LIN {X 0,Y 614.5,Z 958.979,A -85,B 0,C 180,E1 26505.989,E2 26505.989} C_VEL
LIN {X 0,Y 616.34,Z 935.943,A -85,B 0,C 180,E1 26505.389,E2 26505.389} C_VEL
LIN {X 0,Y 618.103,Z 906.869,A -85,B 0,C 180,E1 26504.819,E2 26504.819} C_VEL
LIN {X 0,Y 619.74,Z 852.233,A -85,B 0,C 180,E1 26504.043,E2 26504.043} C_VEL
LIN {X 0,Y 625.607,Z 633.811,A -85,B 0,C 180,E1 26500.991,E2 26500.991} C_VEL
LIN {X 0,Y 629.765,Z 486.938,A -85,B 0,C 180,E1 26498.889,E2 26498.889} C_VEL
LIN {X 0,Y 615.789,Z 466.074,A -85,B 0,C 180,E1 26496.868,E2 26496.868} C_VEL
LIN {X 0,Y 606.821,Z 453.224,A -85,B 0,C 180,E1 26495.48,E2 26495.48} C_VEL
LIN {X 0,Y 598.746,Z 442.127,A -85,B 0,C 180,E1 26494.162,E2 26494.162} C_VEL
LIN {X 0,Y 588.904,Z 428.967,A -85,B 0,C 180,E1 26492.448,E2 26492.448} C_VEL
LIN {X 0,Y 585.376,Z 424.275,A -85,B 0,C 180,E1 26491.8,E2 26491.8} C_VEL
LIN {X 0,Y 583.558,Z 421.917,A -85,B 0,C 180,E1 26491.392,E2 26491.392} C_VEL
LIN {X 0,Y 582.067,Z 418.761,A -85,B 0,C 180,E1 26490.791,E2 26490.791} C_VEL
LIN {X 0,Y 580.207,Z 415.439,A -85,B 0,C 180,E1 26490.099,E2 26490.099} C_VEL
LIN {X 0,Y 579.523,Z 413.86,A -85,B 0,C 180,E1 26489.796,E2 26489.796} C_VEL
LIN {X 0,Y 577.505,Z 410.525,A -85,B 0,C 180,E1 26489.047,E2 26489.047} C_VEL
LIN {X 0,Y 577.246,Z 409.292,A -85,B 0,C 180,E1 26488.795,E2 26488.795} C_VEL
LIN {X 0,Y 577.307,Z 409.275,A -85,B 0,C 180,E1 26485.658,E2 26485.658} C_VEL
LIN {X 0,Y 577.239,Z 409.328,A -85,B 0,C 180,E1 26482.613,E2 26482.613} C_VEL
LIN {X 0,Y 577.304,Z 409.276,A -85,B 0,C 180,E1 26479.529,E2 26479.529} C_VEL
LIN {X 0,Y 577.227,Z 409.31,A -85,B 0,C 180,E1 26476.504,E2 26476.504} C_VEL
LIN {X 0,Y 577.301,Z 409.291,A -85,B 0,C 180,E1 26473.42,E2 26473.42} C_VEL
LIN {X 0,Y 577.214,Z 409.295,A -85,B 0,C 180,E1 26470.278,E2 26470.278} C_VEL
LIN {X 0,Y 577.279,Z 409.308,A -85,B 0,C 180,E1 26467.097,E2 26467.097} C_VEL
LIN {X 0,Y 577.215,Z 409.289,A -85,B 0,C 180,E1 26464.073,E2 26464.073} C_VEL
LIN {X 0,Y 577.286,Z 409.311,A -85,B 0,C 180,E1 26460.893,E2 26460.893} C_VEL
LIN {X 0,Y 577.226,Z 409.286,A -85,B 0,C 180,E1 26457.915,E2 26457.915} C_VEL
LIN {X 0,Y 577.293,Z 409.312,A -85,B 0,C 180,E1 26454.733,E2 26454.733} C_VEL
LIN {X 0,Y 577.237,Z 409.283,A -85,B 0,C 180,E1 26451.734,E2 26451.734} C_VEL
LIN {X 0,Y 577.296,Z 409.318,A -85,B 0,C 180,E1 26448.511,E2 26448.511} C_VEL
LIN {X 0,Y 577.25,Z 409.278,A -85,B 0,C 180,E1 26445.454,E2 26445.454} C_VEL
LIN {X 0,Y 577.285,Z 409.321,A -85,B 0,C 180,E1 26442.147,E2 26442.147} C_VEL
LIN {X 0,Y 577.272,Z 409.275,A -85,B 0,C 180,E1 26439.095,E2 26439.095} C_VEL
LIN {X 0,Y 577.272,Z 409.3,A -85,B 0,C 180,E1 26435.763,E2 26435.763} C_VEL
LIN {X 0,Y 577.315,Z 409.306,A -85,B 0,C 180,E1 26432.567,E2 26432.567} C_VEL
LIN {X 0,Y 577.279,Z 409.351,A -85,B 0,C 180,E1 26429.358,E2 26429.358} C_VEL
LIN {X 0,Y 578.244,Z 412.23,A -85,B 0,C 180,E1 26429.127,E2 26429.127} C_VEL
LIN {X 0,Y 580.66,Z 414.858,A -85,B 0,C 180,E1 26428.665,E2 26428.665} C_VEL
LIN {X 0,Y 582.281,Z 416.079,A -85,B 0,C 180,E1 26428.373,E2 26428.373} C_VEL
LIN {X 0,Y 584.579,Z 419.788,A -85,B 0,C 180,E1 26427.92,E2 26427.92} C_VEL
LIN {X 0,Y 587.298,Z 422.366,A -85,B 0,C 180,E1 26427.438,E2 26427.438} C_VEL
LIN {X 0,Y 590.315,Z 426.389,A -85,B 0,C 180,E1 26426.889,E2 26426.889} C_VEL
LIN {X 0,Y 592.156,Z 428.364,A -85,B 0,C 180,E1 26426.572,E2 26426.572} C_VEL
LIN {X 0,Y 595.83,Z 432.899,A -85,B 0,C 180,E1 26425.938,E2 26425.938} C_VEL
LIN {X 0,Y 602.194,Z 441.085,A -85,B 0,C 180,E1 26424.877,E2 26424.877} C_VEL
LIN {X 0,Y 609.795,Z 450.687,A -85,B 0,C 180,E1 26423.676,E2 26423.676} C_VEL
LIN {X 0,Y 621.483,Z 466.359,A -85,B 0,C 180,E1 26421.931,E2 26421.931} C_VEL
LIN {X 0,Y 629.591,Z 477.801,A -85,B 0,C 180,E1 26420.786,E2 26420.786} C_VEL
LIN {X 0,Y 623.132,Z 702.195,A -85,B 0,C 180,E1 26417.599,E2 26417.599} C_VEL
LIN {X 0,Y 622.882,Z 711.323,A -85,B 0,C 180,E1 26417.471,E2 26417.471} C_VEL
LIN {X 0,Y 621.995,Z 719.027,A -85,B 0,C 180,E1 26417.431,E2 26417.431} C_VEL
LIN {X 0,Y 617.19,Z 739.673,A -85,B 0,C 180,E1 26417.572,E2 26417.572} C_VEL
LIN {X 0,Y 616.501,Z 746.282,A -85,B 0,C 180,E1 26417.53,E2 26417.53} C_VEL
LIN {X 0,Y 612.714,Z 875.215,A -85,B 0,C 180,E1 26415.71,E2 26415.71} C_VEL
LIN {X 0,Y 611.293,Z 900.177,A -85,B 0,C 180,E1 26415.25,E2 26415.25} C_VEL
LIN {X 0,Y 609.06,Z 927.879,A -85,B 0,C 180,E1 26414.552,E2 26414.552} C_VEL
LIN {X 0,Y 606.986,Z 949.44,A -85,B 0,C 180,E1 26413.867,E2 26413.867} C_VEL
LIN {X 0,Y 604.786,Z 969.358,A -85,B 0,C 180,E1 26413.119,E2 26413.119} C_VEL
LIN {X 0,Y 602.352,Z 989.561,A -85,B 0,C 180,E1 26412.235,E2 26412.235} C_VEL
LIN {X 0,Y 599.698,Z 1009.452,A -85,B 0,C 180,E1 26411.239,E2 26411.239} C_VEL
LIN {X 0,Y 596.122,Z 1034.235,A -85,B 0,C 180,E1 26409.806,E2 26409.806} C_VEL
LIN {X 0,Y 592.792,Z 1055.848,A -85,B 0,C 180,E1 26408.361,E2 26408.361} C_VEL
LIN {X 0,Y 589.917,Z 1074.13,A -85,B 0,C 180,E1 26406.985,E2 26406.985} C_VEL
LIN {X 0,Y 587.066,Z 1091.868,A -85,B 0,C 180,E1 26405.498,E2 26405.498} C_VEL
LIN {X 0,Y 583.798,Z 1112.341,A -85,B 0,C 180,E1 26403.58,E2 26403.58} C_VEL
LIN {X 0,Y 580.752,Z 1131.299,A -85,B 0,C 180,E1 26401.542,E2 26401.542} C_VEL
LIN {X 0,Y 578.394,Z 1146.388,A -85,B 0,C 180,E1 26399.738,E2 26399.738} C_VEL
LIN {X 0,Y 576.222,Z 1160.882,A -85,B 0,C 180,E1 26397.819,E2 26397.819} C_VEL
LIN {X 0,Y 573.962,Z 1177.393,A -85,B 0,C 180,E1 26395.369,E2 26395.369} C_VEL
LIN {X 0,Y 572.132,Z 1191.681,A -85,B 0,C 180,E1 26392.924,E2 26392.924} C_VEL
LIN {X 0,Y 570.833,Z 1203.133,A -85,B 0,C 180,E1 26390.711,E2 26390.711} C_VEL
LIN {X 0,Y 569.76,Z 1214.119,A -85,B 0,C 180,E1 26388.3,E2 26388.3} C_VEL
LIN {X 0,Y 568.912,Z 1224.958,A -85,B 0,C 180,E1 26385.489,E2 26385.489} C_VEL
LIN {X 0,Y 568.45,Z 1232.629,A -85,B 0,C 180,E1 26383.11,E2 26383.11} C_VEL
LIN {X 0,Y 568.167,Z 1238.465,A -85,B 0,C 180,E1 26380.951,E2 26380.951} C_VEL
LIN {X 0,Y 568.021,Z 1243.665,A -85,B 0,C 180,E1 26378.6,E2 26378.6} C_VEL
LIN {X 0,Y 567.937,Z 1248.127,A -85,B 0,C 180,E1 26375.856,E2 26375.856} C_VEL
LIN {X 0,Y 567.911,Z 1250.647,A -85,B 0,C 180,E1 26373.326,E2 26373.326} C_VEL
LIN {X 0,Y 567.894,Z 1251.727,A -85,B 0,C 180,E1 26371.206,E2 26371.206} C_VEL
LIN {X 0,Y 567.865,Z 1251.836,A -85,B 0,C 180,E1 26369.188,E2 26369.188} C_VEL
LIN {X 0,Y 567.909,Z 1250.974,A -85,B 0,C 180,E1 26367.069,E2 26367.069} C_VEL
LIN {X 0,Y 567.923,Z 1249.038,A -85,B 0,C 180,E1 26364.844,E2 26364.844} C_VEL
LIN {X 0,Y 567.957,Z 1245.803,A -85,B 0,C 180,E1 26362.51,E2 26362.51} C_VEL
LIN {X 0,Y 568.095,Z 1240.685,A -85,B 0,C 180,E1 26359.859,E2 26359.859} C_VEL
LIN {X 0,Y 568.383,Z 1233.775,A -85,B 0,C 180,E1 26357.19,E2 26357.19} C_VEL
LIN {X 0,Y 568.807,Z 1226.648,A -85,B 0,C 180,E1 26354.916,E2 26354.916} C_VEL
LIN {X 0,Y 569.369,Z 1218.647,A -85,B 0,C 180,E1 26352.732,E2 26352.732} C_VEL
LIN {X 0,Y 570.319,Z 1208.371,A -85,B 0,C 180,E1 26350.302,E2 26350.302} C_VEL
LIN {X 0,Y 571.738,Z 1194.931,A -85,B 0,C 180,E1 26347.585,E2 26347.585} C_VEL
LIN {X 0,Y 573.259,Z 1182.33,A -85,B 0,C 180,E1 26345.36,E2 26345.36} C_VEL
LIN {X 0,Y 575.113,Z 1168.833,A -85,B 0,C 180,E1 26343.234,E2 26343.234} C_VEL
LIN {X 0,Y 577.791,Z 1150.36,A -85,B 0,C 180,E1 26340.673,E2 26340.673} C_VEL
LIN {X 0,Y 580.261,Z 1134.406,A -85,B 0,C 180,E1 26338.726,E2 26338.726} C_VEL
LIN {X 0,Y 582.67,Z 1119.131,A -85,B 0,C 180,E1 26337.041,E2 26337.041} C_VEL
LIN {X 0,Y 585.457,Z 1101.99,A -85,B 0,C 180,E1 26335.336,E2 26335.336} C_VEL
LIN {X 0,Y 588.989,Z 1080.008,A -85,B 0,C 180,E1 26333.391,E2 26333.391} C_VEL
LIN {X 0,Y 592.289,Z 1059.002,A -85,B 0,C 180,E1 26331.775,E2 26331.775} C_VEL
LIN {X 0,Y 595.114,Z 1040.52,A -85,B 0,C 180,E1 26330.507,E2 26330.507} C_VEL
LIN {X 0,Y 598.459,Z 1018.141,A -85,B 0,C 180,E1 26329.145,E2 26329.145} C_VEL
LIN {X 0,Y 602.017,Z 992.189,A -85,B 0,C 180,E1 26327.797,E2 26327.797} C_VEL
LIN {X 0,Y 604.611,Z 970.893,A -85,B 0,C 180,E1 26326.853,E2 26326.853} C_VEL
LIN {X 0,Y 606.877,Z 950.456,A -85,B 0,C 180,E1 26326.078,E2 26326.078} C_VEL
LIN {X 0,Y 608.924,Z 929.275,A -85,B 0,C 180,E1 26325.399,E2 26325.399} C_VEL
LIN {X 0,Y 611.085,Z 903.304,A -85,B 0,C 180,E1 26324.725,E2 26324.725} C_VEL
LIN {X 0,Y 612.671,Z 876.135,A -85,B 0,C 180,E1 26324.214,E2 26324.214} C_VEL
LIN {X 0,Y 615.283,Z 789.302,A -85,B 0,C 180,E1 26322.984,E2 26322.984} C_VEL
LIN {X 0,Y 621.588,Z 573.63,A -85,B 0,C 180,E1 26319.929,E2 26319.929} C_VEL
LIN {X 0,Y 624.375,Z 481.675,A -85,B 0,C 180,E1 26318.597,E2 26318.597} C_VEL
LIN {X 0,Y 611.48,Z 463.889,A -85,B 0,C 180,E1 26316.703,E2 26316.703} C_VEL
LIN {X 0,Y 600.781,Z 449.867,A -85,B 0,C 180,E1 26315.014,E2 26315.014} C_VEL
LIN {X 0,Y 592.208,Z 439.07,A -85,B 0,C 180,E1 26313.57,E2 26313.57} C_VEL
LIN {X 0,Y 587.983,Z 433.825,A -85,B 0,C 180,E1 26312.823,E2 26312.823} C_VEL
LIN {X 0,Y 584.443,Z 429.323,A -85,B 0,C 180,E1 26312.175,E2 26312.175} C_VEL
LIN {X 0,Y 580.339,Z 424.729,A -85,B 0,C 180,E1 26311.412,E2 26311.412} C_VEL
LIN {X 0,Y 579.006,Z 422.68,A -85,B 0,C 180,E1 26311.145,E2 26311.145} C_VEL
LIN {X 0,Y 575.874,Z 419.674,A -85,B 0,C 180,E1 26310.549,E2 26310.549} C_VEL
LIN {X 0,Y 574.075,Z 416.59,A -85,B 0,C 180,E1 26310.165,E2 26310.165} C_VEL
LIN {X 0,Y 571.098,Z 414.334,A -85,B 0,C 180,E1 26309.586,E2 26309.586} C_VEL
LIN {X 0,Y 569.594,Z 411.434,A -85,B 0,C 180,E1 26309.243,E2 26309.243} C_VEL
LIN {X 0,Y 569.366,Z 410.274,A -85,B 0,C 180,E1 26309.159,E2 26309.159} C_VEL
LIN {X 0,Y 569.371,Z 410.259,A -85,B 0,C 180,E1 26305.819,E2 26305.819} C_VEL
LIN {X 0,Y 569.375,Z 410.302,A -85,B 0,C 180,E1 26302.509,E2 26302.509} C_VEL
LIN {X 0,Y 569.357,Z 410.273,A -85,B 0,C 180,E1 26299.172,E2 26299.172} C_VEL
LIN {X 0,Y 569.367,Z 410.272,A -85,B 0,C 180,E1 26296.005,E2 26296.005} C_VEL
LIN {X 0,Y 569.357,Z 410.297,A -85,B 0,C 180,E1 26292.784,E2 26292.784} C_VEL
LIN {X 0,Y 569.369,Z 410.256,A -85,B 0,C 180,E1 26289.502,E2 26289.502} C_VEL
LIN {X 0,Y 569.375,Z 410.305,A -85,B 0,C 180,E1 26286.15,E2 26286.15} C_VEL
LIN {X 0,Y 569.351,Z 410.252,A -85,B 0,C 180,E1 26282.718,E2 26282.718} C_VEL
LIN {X 0,Y 569.375,Z 410.306,A -85,B 0,C 180,E1 26279.497,E2 26279.497} C_VEL
LIN {X 0,Y 569.347,Z 410.254,A -85,B 0,C 180,E1 26276.173,E2 26276.173} C_VEL
LIN {X 0,Y 569.385,Z 410.296,A -85,B 0,C 180,E1 26272.838,E2 26272.838} C_VEL
LIN {X 0,Y 569.368,Z 410.268,A -85,B 0,C 180,E1 26269.476,E2 26269.476} C_VEL
LIN {X 0,Y 569.351,Z 410.273,A -85,B 0,C 180,E1 26266.182,E2 26266.182} C_VEL
LIN {X 0,Y 569.378,Z 410.298,A -85,B 0,C 180,E1 26262.946,E2 26262.946} C_VEL
LIN {X 0,Y 569.343,Z 410.261,A -85,B 0,C 180,E1 26259.651,E2 26259.651} C_VEL
LIN {X 0,Y 569.379,Z 410.289,A -85,B 0,C 180,E1 26256.397,E2 26256.397} C_VEL
LIN {X 0,Y 569.351,Z 410.29,A -85,B 0,C 180,E1 26253.148,E2 26253.148} C_VEL
LIN {X 0,Y 569.4,Z 410.443,A -85,B 0,C 180,E1 26252.412,E2 26252.412} C_VEL
LIN {X 0,Y 570.618,Z 413.713,A -85,B 0,C 180,E1 26251.763,E2 26251.763} C_VEL
LIN {X 0,Y 572.078,Z 415.531,A -85,B 0,C 180,E1 26251.272,E2 26251.272} C_VEL
LIN {X 0,Y 573.957,Z 419.421,A -85,B 0,C 180,E1 26250.461,E2 26250.461} C_VEL
LIN {X 0,Y 574.968,Z 421.314,A -85,B 0,C 180,E1 26250.059,E2 26250.059} C_VEL
LIN {X 0,Y 576.403,Z 423.685,A -85,B 0,C 180,E1 26249.682,E2 26249.682} C_VEL
LIN {X 0,Y 579.802,Z 427.922,A -85,B 0,C 180,E1 26249.017,E2 26249.017} C_VEL
LIN {X 0,Y 583.259,Z 432.351,A -85,B 0,C 180,E1 26248.36,E2 26248.36} C_VEL
LIN {X 0,Y 587.845,Z 438.306,A -85,B 0,C 180,E1 26247.515,E2 26247.515} C_VEL
LIN {X 0,Y 598.795,Z 453.112,A -85,B 0,C 180,E1 26245.61,E2 26245.61} C_VEL
LIN {X 0,Y 609.202,Z 467.887,A -85,B 0,C 180,E1 26243.926,E2 26243.926} C_VEL
LIN {X 0,Y 619.523,Z 483.235,A -85,B 0,C 180,E1 26242.361,E2 26242.361} C_VEL
LIN {X 0,Y 624.656,Z 491.339,A -85,B 0,C 180,E1 26241.613,E2 26241.613} C_VEL
LIN {X 0,Y 618.21,Z 707.468,A -85,B 0,C 180,E1 26238.522,E2 26238.522} C_VEL
LIN {X 0,Y 612.621,Z 902.713,A -85,B 0,C 180,E1 26235.775,E2 26235.775} C_VEL
LIN {X 0,Y 611.268,Z 926.421,A -85,B 0,C 180,E1 26235.348,E2 26235.348} C_VEL
LIN {X 0,Y 609.018,Z 955.255,A -85,B 0,C 180,E1 26234.642,E2 26234.642} C_VEL
LIN {X 0,Y 606.904,Z 977.493,A -85,B 0,C 180,E1 26233.948,E2 26233.948} C_VEL
LIN {X 0,Y 604.637,Z 998.395,A -85,B 0,C 180,E1 26233.173,E2 26233.173} C_VEL
LIN {X 0,Y 602.31,Z 1018.258,A -85,B 0,C 180,E1 26232.315,E2 26232.315} C_VEL
LIN {X 0,Y 599.707,Z 1038.412,A -85,B 0,C 180,E1 26231.322,E2 26231.322} C_VEL
LIN {X 0,Y 596.389,Z 1062.63,A -85,B 0,C 180,E1 26229.953,E2 26229.953} C_VEL
LIN {X 0,Y 592.85,Z 1085.526,A -85,B 0,C 180,E1 26228.429,E2 26228.429} C_VEL
LIN {X 0,Y 589.917,Z 1104.147,A -85,B 0,C 180,E1 26227.029,E2 26227.029} C_VEL
LIN {X 0,Y 587.11,Z 1121.609,A -85,B 0,C 180,E1 26225.566,E2 26225.566} C_VEL
LIN {X 0,Y 583.857,Z 1141.944,A -85,B 0,C 180,E1 26223.663,E2 26223.663} C_VEL
LIN {X 0,Y 580.67,Z 1161.802,A -85,B 0,C 180,E1 26221.529,E2 26221.529} C_VEL
LIN {X 0,Y 578.358,Z 1176.644,A -85,B 0,C 180,E1 26219.751,E2 26219.751} C_VEL
LIN {X 0,Y 576.185,Z 1191.121,A -85,B 0,C 180,E1 26217.831,E2 26217.831} C_VEL
LIN {X 0,Y 573.932,Z 1207.596,A -85,B 0,C 180,E1 26215.381,E2 26215.381} C_VEL
LIN {X 0,Y 572.091,Z 1221.975,A -85,B 0,C 180,E1 26212.915,E2 26212.915} C_VEL
LIN {X 0,Y 570.807,Z 1233.381,A -85,B 0,C 180,E1 26210.704,E2 26210.704} C_VEL
LIN {X 0,Y 569.687,Z 1245.179,A -85,B 0,C 180,E1 26208.103,E2 26208.103} C_VEL
LIN {X 0,Y 568.881,Z 1255.436,A -85,B 0,C 180,E1 26205.395,E2 26205.395} C_VEL
LIN {X 0,Y 568.444,Z 1262.734,A -85,B 0,C 180,E1 26203.119,E2 26203.119} C_VEL
LIN {X 0,Y 568.156,Z 1268.75,A -85,B 0,C 180,E1 26200.881,E2 26200.881} C_VEL
LIN {X 0,Y 568.007,Z 1274.19,A -85,B 0,C 180,E1 26198.381,E2 26198.381} C_VEL
LIN {X 0,Y 567.927,Z 1278.533,A -85,B 0,C 180,E1 26195.561,E2 26195.561} C_VEL
LIN {X 0,Y 567.911,Z 1280.74,A -85,B 0,C 180,E1 26193.234,E2 26193.234} C_VEL
LIN {X 0,Y 567.889,Z 1281.735,A -85,B 0,C 180,E1 26191.215,E2 26191.215} C_VEL
LIN {X 0,Y 567.865,Z 1281.828,A -85,B 0,C 180,E1 26189.198,E2 26189.198} C_VEL
LIN {X 0,Y 567.91,Z 1281.018,A -85,B 0,C 180,E1 26187.179,E2 26187.179} C_VEL
LIN {X 0,Y 567.922,Z 1279.111,A -85,B 0,C 180,E1 26184.955,E2 26184.955} C_VEL
LIN {X 0,Y 567.957,Z 1275.906,A -85,B 0,C 180,E1 26182.621,E2 26182.621} C_VEL
LIN {X 0,Y 568.069,Z 1271.048,A -85,B 0,C 180,E1 26180.072,E2 26180.072} C_VEL
LIN {X 0,Y 568.368,Z 1263.973,A -85,B 0,C 180,E1 26177.302,E2 26177.302} C_VEL
LIN {X 0,Y 568.791,Z 1256.879,A -85,B 0,C 180,E1 26175.03,E2 26175.03} C_VEL
LIN {X 0,Y 569.351,Z 1248.811,A -85,B 0,C 180,E1 26172.818,E2 26172.818} C_VEL
LIN {X 0,Y 570.275,Z 1238.792,A -85,B 0,C 180,E1 26170.44,E2 26170.44} C_VEL
LIN {X 0,Y 571.693,Z 1225.323,A -85,B 0,C 180,E1 26167.702,E2 26167.702} C_VEL
LIN {X 0,Y 573.202,Z 1212.765,A -85,B 0,C 180,E1 26165.477,E2 26165.477} C_VEL
LIN {X 0,Y 575.049,Z 1199.284,A -85,B 0,C 180,E1 26163.347,E2 26163.347} C_VEL
LIN {X 0,Y 577.58,Z 1181.792,A -85,B 0,C 180,E1 26160.899,E2 26160.899} C_VEL
LIN {X 0,Y 580.196,Z 1164.81,A -85,B 0,C 180,E1 26158.818,E2 26158.818} C_VEL
LIN {X 0,Y 582.638,Z 1149.342,A -85,B 0,C 180,E1 26157.109,E2 26157.109} C_VEL
LIN {X 0,Y 585.394,Z 1132.354,A -85,B 0,C 180,E1 26155.416,E2 26155.416} C_VEL
LIN {X 0,Y 588.897,Z 1110.634,A -85,B 0,C 180,E1 26153.487,E2 26153.487} C_VEL
LIN {X 0,Y 592.234,Z 1089.323,A -85,B 0,C 180,E1 26151.843,E2 26151.843} C_VEL
LIN {X 0,Y 595.18,Z 1070.076,A -85,B 0,C 180,E1 26150.524,E2 26150.524} C_VEL
LIN {X 0,Y 597.856,Z 1051.647,A -85,B 0,C 180,E1 26149.403,E2 26149.403} C_VEL
LIN {X 0,Y 601.021,Z 1028.469,A -85,B 0,C 180,E1 26148.163,E2 26148.163} C_VEL
LIN {X 0,Y 604.116,Z 1003.087,A -85,B 0,C 180,E1 26147.016,E2 26147.016} C_VEL
LIN {X 0,Y 606.495,Z 981.393,A -85,B 0,C 180,E1 26146.187,E2 26146.187} C_VEL
LIN {X 0,Y 608.555,Z 960.121,A -85,B 0,C 180,E1 26145.499,E2 26145.499} C_VEL
LIN {X 0,Y 610.366,Z 938.714,A -85,B 0,C 180,E1 26144.93,E2 26144.93} C_VEL
LIN {X 0,Y 611.998,Z 915.01,A -85,B 0,C 180,E1 26144.429,E2 26144.429} C_VEL
LIN {X 0,Y 613.45,Z 878.801,A -85,B 0,C 180,E1 26143.877,E2 26143.877} C_VEL
LIN {X 0,Y 619.746,Z 654.48,A -85,B 0,C 180,E1 26140.728,E2 26140.728} C_VEL
LIN {X 0,Y 624.575,Z 490.916,A -85,B 0,C 180,E1 26138.371,E2 26138.371} C_VEL
LIN {X 0,Y 611.652,Z 471.495,A -85,B 0,C 180,E1 26136.458,E2 26136.458} C_VEL
LIN {X 0,Y 602.911,Z 458.902,A -85,B 0,C 180,E1 26135.075,E2 26135.075} C_VEL
LIN {X 0,Y 593.469,Z 445.801,A -85,B 0,C 180,E1 26133.489,E2 26133.489} C_VEL
LIN {X 0,Y 585.554,Z 435.346,A -85,B 0,C 180,E1 26132.077,E2 26132.077} C_VEL
LIN {X 0,Y 580.441,Z 428.74,A -85,B 0,C 180,E1 26131.117,E2 26131.117} C_VEL
LIN {X 0,Y 575.132,Z 421.811,A -85,B 0,C 180,E1 26130.042,E2 26130.042} C_VEL
LIN {X 0,Y 574.226,Z 419.751,A -85,B 0,C 180,E1 26129.639,E2 26129.639} C_VEL
LIN {X 0,Y 572.185,Z 416.114,A -85,B 0,C 180,E1 26128.836,E2 26128.836} C_VEL
LIN {X 0,Y 571.43,Z 414.783,A -85,B 0,C 180,E1 26128.535,E2 26128.535} C_VEL
LIN {X 0,Y 569.662,Z 411.624,A -85,B 0,C 180,E1 26127.809,E2 26127.809} C_VEL
LIN {X 0,Y 569.362,Z 410.311,A -85,B 0,C 180,E1 26127.535,E2 26127.535} C_VEL
LIN {X 0,Y 569.302,Z 410.274,A -85,B 0,C 180,E1 26124.488,E2 26124.488} C_VEL
LIN {X 0,Y 569.329,Z 410.273,A -85,B 0,C 180,E1 26121.21,E2 26121.21} C_VEL
LIN {X 0,Y 569.304,Z 410.309,A -85,B 0,C 180,E1 26118.187,E2 26118.187} C_VEL
LIN {X 0,Y 569.29,Z 410.266,A -85,B 0,C 180,E1 26114.754,E2 26114.754} C_VEL
LIN {X 0,Y 569.306,Z 410.317,A -85,B 0,C 180,E1 26111.858,E2 26111.858} C_VEL
LIN {X 0,Y 569.278,Z 410.269,A -85,B 0,C 180,E1 26108.586,E2 26108.586} C_VEL
LIN {X 0,Y 569.297,Z 410.318,A -85,B 0,C 180,E1 26105.746,E2 26105.746} C_VEL
LIN {X 0,Y 569.285,Z 410.269,A -85,B 0,C 180,E1 26102.416,E2 26102.416} C_VEL
LIN {X 0,Y 569.314,Z 410.311,A -85,B 0,C 180,E1 26099.497,E2 26099.497} C_VEL
LIN {X 0,Y 569.293,Z 410.27,A -85,B 0,C 180,E1 26096.173,E2 26096.173} C_VEL
LIN {X 0,Y 569.346,Z 410.3,A -85,B 0,C 180,E1 26093.141,E2 26093.141} C_VEL
LIN {X 0,Y 569.301,Z 410.274,A -85,B 0,C 180,E1 26089.884,E2 26089.884} C_VEL
LIN {X 0,Y 569.381,Z 410.283,A -85,B 0,C 180,E1 26086.7,E2 26086.7} C_VEL
LIN {X 0,Y 569.311,Z 410.286,A -85,B 0,C 180,E1 26083.574,E2 26083.574} C_VEL
LIN {X 0,Y 569.375,Z 410.264,A -85,B 0,C 180,E1 26080.402,E2 26080.402} C_VEL
LIN {X 0,Y 569.331,Z 410.311,A -85,B 0,C 180,E1 26077.205,E2 26077.205} C_VEL
LIN {X 0,Y 569.341,Z 410.266,A -85,B 0,C 180,E1 26073.805,E2 26073.805} C_VEL
LIN {X 0,Y 569.393,Z 410.514,A -85,B 0,C 180,E1 26070.711,E2 26070.711} C_VEL
LIN {X 0,Y 570.498,Z 413.457,A -85,B 0,C 180,E1 26070.437,E2 26070.437} C_VEL
LIN {X 0,Y 572.942,Z 415.978,A -85,B 0,C 180,E1 26069.942,E2 26069.942} C_VEL
LIN {X 0,Y 574.39,Z 417.026,A -85,B 0,C 180,E1 26069.665,E2 26069.665} C_VEL
LIN {X 0,Y 576.595,Z 420.637,A -85,B 0,C 180,E1 26069.203,E2 26069.203} C_VEL
LIN {X 0,Y 579.568,Z 423.425,A -85,B 0,C 180,E1 26068.642,E2 26068.642} C_VEL
LIN {X 0,Y 582.588,Z 427.545,A -85,B 0,C 180,E1 26068.059,E2 26068.059} C_VEL
LIN {X 0,Y 584.614,Z 429.641,A -85,B 0,C 180,E1 26067.691,E2 26067.691} C_VEL
LIN {X 0,Y 588.179,Z 433.994,A -85,B 0,C 180,E1 26067.044,E2 26067.044} C_VEL
LIN {X 0,Y 594.983,Z 442.6,A -85,B 0,C 180,E1 26065.854,E2 26065.854} C_VEL
LIN {X 0,Y 599.346,Z 448.153,A -85,B 0,C 180,E1 26065.123,E2 26065.123} C_VEL
LIN {X 0,Y 607.404,Z 458.511,A -85,B 0,C 180,E1 26063.832,E2 26063.832} C_VEL
LIN {X 0,Y 618.096,Z 472.942,A -85,B 0,C 180,E1 26062.215,E2 26062.215} C_VEL
LIN {X 0,Y 624.433,Z 481.944,A -85,B 0,C 180,E1 26061.3,E2 26061.3} C_VEL
LIN {X 0,Y 617.707,Z 704.407,A -85,B 0,C 180,E1 26058.12,E2 26058.12} C_VEL
LIN {X 0,Y 616.501,Z 746.282,A -85,B 0,C 180,E1 26057.53,E2 26057.53} C_VEL
LIN {X 0,Y 615.615,Z 753.984,A -85,B 0,C 180,E1 26057.49,E2 26057.49} C_VEL
LIN {X 0,Y 610.794,Z 774.622,A -85,B 0,C 180,E1 26057.635,E2 26057.635} C_VEL
LIN {X 0,Y 610.089,Z 781.231,A -85,B 0,C 180,E1 26057.594,E2 26057.594} C_VEL
LIN {X 0,Y 607.124,Z 876.158,A -85,B 0,C 180,E1 26056.241,E2 26056.241} C_VEL
LIN {X 0,Y 605.504,Z 903.148,A -85,B 0,C 180,E1 26055.733,E2 26055.733} C_VEL
LIN {X 0,Y 603.235,Z 929.375,A -85,B 0,C 180,E1 26055.052,E2 26055.052} C_VEL
LIN {X 0,Y 601.115,Z 950.458,A -85,B 0,C 180,E1 26054.374,E2 26054.374} C_VEL
LIN {X 0,Y 598.748,Z 970.915,A -85,B 0,C 180,E1 26053.597,E2 26053.597} C_VEL
LIN {X 0,Y 596.068,Z 992.084,A -85,B 0,C 180,E1 26052.655,E2 26052.655} C_VEL
LIN {X 0,Y 592.485,Z 1017.319,A -85,B 0,C 180,E1 26051.345,E2 26051.345} C_VEL
LIN {X 0,Y 589.093,Z 1038.901,A -85,B 0,C 180,E1 26050.029,E2 26050.029} C_VEL
LIN {X 0,Y 586.068,Z 1057.34,A -85,B 0,C 180,E1 26048.757,E2 26048.757} C_VEL
LIN {X 0,Y 583.065,Z 1075.471,A -85,B 0,C 180,E1 26047.37,E2 26047.37} C_VEL
LIN {X 0,Y 579.804,Z 1094.76,A -85,B 0,C 180,E1 26045.722,E2 26045.722} C_VEL
LIN {X 0,Y 576.048,Z 1116.772,A -85,B 0,C 180,E1 26043.573,E2 26043.573} C_VEL
LIN {X 0,Y 573.311,Z 1133.066,A -85,B 0,C 180,E1 26041.776,E2 26041.776} C_VEL
LIN {X 0,Y 570.841,Z 1148.081,A -85,B 0,C 180,E1 26039.94,E2 26039.94} C_VEL
LIN {X 0,Y 568.118,Z 1165.498,A -85,B 0,C 180,E1 26037.566,E2 26037.566} C_VEL
LIN {X 0,Y 565.821,Z 1181.237,A -85,B 0,C 180,E1 26035.088,E2 26035.088} C_VEL
LIN {X 0,Y 564.227,Z 1193.368,A -85,B 0,C 180,E1 26032.94,E2 26032.94} C_VEL
LIN {X 0,Y 562.798,Z 1205.685,A -85,B 0,C 180,E1 26030.481,E2 26030.481} C_VEL
LIN {X 0,Y 561.6,Z 1217.53,A -85,B 0,C 180,E1 26027.719,E2 26027.719} C_VEL
LIN {X 0,Y 560.918,Z 1226.022,A -85,B 0,C 180,E1 26025.397,E2 26025.397} C_VEL
LIN {X 0,Y 560.457,Z 1233.301,A -85,B 0,C 180,E1 26023.068,E2 26023.068} C_VEL
LIN {X 0,Y 560.156,Z 1239.737,A -85,B 0,C 180,E1 26020.589,E2 26020.589} C_VEL
LIN {X 0,Y 559.958,Z 1245.354,A -85,B 0,C 180,E1 26017.794,E2 26017.794} C_VEL
LIN {X 0,Y 559.925,Z 1248.831,A -85,B 0,C 180,E1 26015.323,E2 26015.323} C_VEL
LIN {X 0,Y 559.91,Z 1250.852,A -85,B 0,C 180,E1 26013.066,E2 26013.066} C_VEL
LIN {X 0,Y 559.88,Z 1251.772,A -85,B 0,C 180,E1 26011.019,E2 26011.019} C_VEL
LIN {X 0,Y 559.873,Z 1251.79,A -85,B 0,C 180,E1 26008.972,E2 26008.972} C_VEL
LIN {X 0,Y 559.91,Z 1250.906,A -85,B 0,C 180,E1 26006.924,E2 26006.924} C_VEL
LIN {X 0,Y 559.923,Z 1248.921,A -85,B 0,C 180,E1 26004.667,E2 26004.667} C_VEL
LIN {X 0,Y 559.961,Z 1245.479,A -85,B 0,C 180,E1 26002.196,E2 26002.196} C_VEL
LIN {X 0,Y 560.149,Z 1239.934,A -85,B 0,C 180,E1 25999.401,E2 25999.401} C_VEL
LIN {X 0,Y 560.448,Z 1233.47,A -85,B 0,C 180,E1 25996.9,E2 25996.9} C_VEL
LIN {X 0,Y 560.897,Z 1226.292,A -85,B 0,C 180,E1 25994.593,E2 25994.593} C_VEL
LIN {X 0,Y 561.575,Z 1217.833,A -85,B 0,C 180,E1 25992.27,E2 25992.27} C_VEL
LIN {X 0,Y 562.806,Z 1205.544,A -85,B 0,C 180,E1 25989.401,E2 25989.401} C_VEL
LIN {X 0,Y 564.173,Z 1193.778,A -85,B 0,C 180,E1 25987.048,E2 25987.048} C_VEL
LIN {X 0,Y 565.754,Z 1181.688,A -85,B 0,C 180,E1 25984.899,E2 25984.899} C_VEL
LIN {X 0,Y 567.927,Z 1166.71,A -85,B 0,C 180,E1 25982.527,E2 25982.527} C_VEL
LIN {X 0,Y 570.623,Z 1149.506,A -85,B 0,C 180,E1 25980.152,E2 25980.152} C_VEL
LIN {X 0,Y 573.132,Z 1134.152,A -85,B 0,C 180,E1 25978.261,E2 25978.261} C_VEL
LIN {X 0,Y 575.729,Z 1118.616,A -85,B 0,C 180,E1 25976.533,E2 25976.533} C_VEL
LIN {X 0,Y 578.957,Z 1099.761,A -85,B 0,C 180,E1 25974.647,E2 25974.647} C_VEL
LIN {X 0,Y 582.695,Z 1077.665,A -85,B 0,C 180,E1 25972.715,E2 25972.715} C_VEL
LIN {X 0,Y 585.812,Z 1058.869,A -85,B 0,C 180,E1 25971.264,E2 25971.264} C_VEL
LIN {X 0,Y 588.833,Z 1040.453,A -85,B 0,C 180,E1 25969.982,E2 25969.982} C_VEL
LIN {X 0,Y 591.866,Z 1021.076,A -85,B 0,C 180,E1 25968.784,E2 25968.784} C_VEL
LIN {X 0,Y 595.457,Z 996.787,A -85,B 0,C 180,E1 25967.475,E2 25967.475} C_VEL
LIN {X 0,Y 598.571,Z 972.42,A -85,B 0,C 180,E1 25966.375,E2 25966.375} C_VEL
LIN {X 0,Y 600.925,Z 952.174,A -85,B 0,C 180,E1 25965.596,E2 25965.596} C_VEL
LIN {X 0,Y 603.043,Z 931.352,A -85,B 0,C 180,E1 25964.917,E2 25964.917} C_VEL
LIN {X 0,Y 604.949,Z 909.636,A -85,B 0,C 180,E1 25964.335,E2 25964.335} C_VEL
LIN {X 0,Y 606.818,Z 883.158,A -85,B 0,C 180,E1 25963.78,E2 25963.78} C_VEL
LIN {X 0,Y 608.39,Z 839.32,A -85,B 0,C 180,E1 25963.134,E2 25963.134} C_VEL
LIN {X 0,Y 615.077,Z 618.061,A -85,B 0,C 180,E1 25959.994,E2 25959.994} C_VEL
LIN {X 0,Y 619.307,Z 485.889,A -85,B 0,C 180,E1 25958.079,E2 25958.079} C_VEL
LIN {X 0,Y 605.577,Z 466.926,A -85,B 0,C 180,E1 25956.002,E2 25956.002} C_VEL
LIN {X 0,Y 593.71,Z 451.476,A -85,B 0,C 180,E1 25954.054,E2 25954.054} C_VEL
LIN {X 0,Y 588.215,Z 444.699,A -85,B 0,C 180,E1 25953.099,E2 25953.099} C_VEL
LIN {X 0,Y 584.879,Z 440.491,A -85,B 0,C 180,E1 25952.496,E2 25952.496} C_VEL
LIN {X 0,Y 580.547,Z 435.165,A -85,B 0,C 180,E1 25951.689,E2 25951.689} C_VEL
LIN {X 0,Y 577.001,Z 430.766,A -85,B 0,C 180,E1 25951.005,E2 25951.005} C_VEL
LIN {X 0,Y 575.281,Z 428.961,A -85,B 0,C 180,E1 25950.673,E2 25950.673} C_VEL
LIN {X 0,Y 572.178,Z 425.064,A -85,B 0,C 180,E1 25950.044,E2 25950.044} C_VEL
LIN {X 0,Y 571.322,Z 423.781,A -85,B 0,C 180,E1 25949.862,E2 25949.862} C_VEL
LIN {X 0,Y 568.196,Z 420.938,A -85,B 0,C 180,E1 25949.231,E2 25949.231} C_VEL
LIN {X 0,Y 566.375,Z 417.698,A -85,B 0,C 180,E1 25948.814,E2 25948.814} C_VEL
LIN {X 0,Y 563.399,Z 415.624,A -85,B 0,C 180,E1 25948.199,E2 25948.199} C_VEL
LIN {X 0,Y 561.737,Z 412.68,A -85,B 0,C 180,E1 25947.798,E2 25947.798} C_VEL
LIN {X 0,Y 561.435,Z 411.294,A -85,B 0,C 180,E1 25947.699,E2 25947.699} C_VEL
LIN {X 0,Y 561.427,Z 411.259,A -85,B 0,C 180,E1 25944.405,E2 25944.405} C_VEL
LIN {X 0,Y 561.418,Z 411.253,A -85,B 0,C 180,E1 25941.195,E2 25941.195} C_VEL
LIN {X 0,Y 561.437,Z 411.297,A -85,B 0,C 180,E1 25937.838,E2 25937.838} C_VEL
LIN {X 0,Y 561.435,Z 411.242,A -85,B 0,C 180,E1 25934.438,E2 25934.438} C_VEL
LIN {X 0,Y 561.424,Z 411.288,A -85,B 0,C 180,E1 25931.084,E2 25931.084} C_VEL
LIN {X 0,Y 561.431,Z 411.25,A -85,B 0,C 180,E1 25927.779,E2 25927.779} C_VEL
LIN {X 0,Y 561.413,Z 411.273,A -85,B 0,C 180,E1 25924.597,E2 25924.597} C_VEL
LIN {X 0,Y 561.436,Z 411.26,A -85,B 0,C 180,E1 25921.225,E2 25921.225} C_VEL
LIN {X 0,Y 561.42,Z 411.255,A -85,B 0,C 180,E1 25917.959,E2 25917.959} C_VEL
LIN {X 0,Y 561.422,Z 411.282,A -85,B 0,C 180,E1 25914.584,E2 25914.584} C_VEL
LIN {X 0,Y 561.435,Z 411.243,A -85,B 0,C 180,E1 25911.396,E2 25911.396} C_VEL
LIN {X 0,Y 561.412,Z 411.296,A -85,B 0,C 180,E1 25908.077,E2 25908.077} C_VEL
LIN {X 0,Y 561.433,Z 411.243,A -85,B 0,C 180,E1 25904.823,E2 25904.823} C_VEL
LIN {X 0,Y 561.413,Z 411.281,A -85,B 0,C 180,E1 25901.517,E2 25901.517} C_VEL
LIN {X 0,Y 561.426,Z 411.273,A -85,B 0,C 180,E1 25898.113,E2 25898.113} C_VEL
LIN {X 0,Y 561.433,Z 411.247,A -85,B 0,C 180,E1 25894.79,E2 25894.79} C_VEL
LIN {X 0,Y 561.438,Z 411.446,A -85,B 0,C 180,E1 25893.789,E2 25893.789} C_VEL
LIN {X 0,Y 562.772,Z 414.837,A -85,B 0,C 180,E1 25893.059,E2 25893.059} C_VEL
LIN {X 0,Y 564.213,Z 416.489,A -85,B 0,C 180,E1 25892.563,E2 25892.563} C_VEL
LIN {X 0,Y 565.931,Z 420.339,A -85,B 0,C 180,E1 25891.738,E2 25891.738} C_VEL
LIN {X 0,Y 567.162,Z 422.075,A -85,B 0,C 180,E1 25891.345,E2 25891.345} C_VEL
LIN {X 0,Y 570.592,Z 426.513,A -85,B 0,C 180,E1 25890.616,E2 25890.616} C_VEL
LIN {X 0,Y 580.096,Z 438.741,A -85,B 0,C 180,E1 25888.718,E2 25888.718} C_VEL
LIN {X 0,Y 588.785,Z 450.227,A -85,B 0,C 180,E1 25887.111,E2 25887.111} C_VEL
LIN {X 0,Y 599.312,Z 464.911,A -85,B 0,C 180,E1 25885.296,E2 25885.296} C_VEL
LIN {X 0,Y 611.079,Z 482.011,A -85,B 0,C 180,E1 25883.415,E2 25883.415} C_VEL
LIN {X 0,Y 619.542,Z 495.336,A -85,B 0,C 180,E1 25882.135,E2 25882.135} C_VEL
LIN {X 0,Y 612.7,Z 713.872,A -85,B 0,C 180,E1 25878.992,E2 25878.992} C_VEL
LIN {X 0,Y 607.025,Z 902.595,A -85,B 0,C 180,E1 25876.317,E2 25876.317} C_VEL
LIN {X 0,Y 605.589,Z 926.645,A -85,B 0,C 180,E1 25875.881,E2 25875.881} C_VEL
LIN {X 0,Y 603.24,Z 955.315,A -85,B 0,C 180,E1 25875.174,E2 25875.174} C_VEL
LIN {X 0,Y 601.069,Z 977.131,A -85,B 0,C 180,E1 25874.491,E2 25874.491} C_VEL
LIN {X 0,Y 598.673,Z 998.243,A -85,B 0,C 180,E1 25873.705,E2 25873.705} C_VEL
LIN {X 0,Y 596.264,Z 1017.874,A -85,B 0,C 180,E1 25872.852,E2 25872.852} C_VEL
LIN {X 0,Y 593.512,Z 1038.14,A -85,B 0,C 180,E1 25871.85,E2 25871.85} C_VEL
LIN {X 0,Y 589.916,Z 1063.108,A -85,B 0,C 180,E1 25870.425,E2 25870.425} C_VEL
LIN {X 0,Y 586.383,Z 1085.428,A -85,B 0,C 180,E1 25868.938,E2 25868.938} C_VEL
LIN {X 0,Y 583.458,Z 1103.173,A -85,B 0,C 180,E1 25867.599,E2 25867.599} C_VEL
LIN {X 0,Y 580.564,Z 1120.302,A -85,B 0,C 180,E1 25866.16,E2 25866.16} C_VEL
LIN {X 0,Y 577.698,Z 1137.118,A -85,B 0,C 180,E1 25864.594,E2 25864.594} C_VEL
LIN {X 0,Y 574.382,Z 1156.838,A -85,B 0,C 180,E1 25862.545,E2 25862.545} C_VEL
LIN {X 0,Y 571.301,Z 1175.145,A -85,B 0,C 180,E1 25860.362,E2 25860.362} C_VEL
LIN {X 0,Y 569.028,Z 1189.578,A -85,B 0,C 180,E1 25858.441,E2 25858.441} C_VEL
LIN {X 0,Y 566.898,Z 1203.649,A -85,B 0,C 180,E1 25856.361,E2 25856.361} C_VEL
LIN {X 0,Y 564.729,Z 1219.523,A -85,B 0,C 180,E1 25853.702,E2 25853.702} C_VEL
LIN {X 0,Y 563.205,Z 1231.728,A -85,B 0,C 180,E1 25851.346,E2 25851.346} C_VEL
LIN {X 0,Y 562.128,Z 1241.685,A -85,B 0,C 180,E1 25849.174,E2 25849.174} C_VEL
LIN {X 0,Y 561.298,Z 1250.904,A -85,B 0,C 180,E1 25846.884,E2 25846.884} C_VEL
LIN {X 0,Y 560.576,Z 1260.603,A -85,B 0,C 180,E1 25844.043,E2 25844.043} C_VEL
LIN {X 0,Y 560.232,Z 1267.567,A -85,B 0,C 180,E1 25841.522,E2 25841.522} C_VEL
LIN {X 0,Y 560.015,Z 1272.495,A -85,B 0,C 180,E1 25839.355,E2 25839.355} C_VEL
LIN {X 0,Y 559.962,Z 1276.528,A -85,B 0,C 180,E1 25837.082,E2 25837.082} C_VEL
LIN {X 0,Y 559.917,Z 1279.667,A -85,B 0,C 180,E1 25834.614,E2 25834.614} C_VEL
LIN {X 0,Y 559.909,Z 1281.622,A -85,B 0,C 180,E1 25831.744,E2 25831.744} C_VEL
LIN {X 0,Y 559.865,Z 1281.873,A -85,B 0,C 180,E1 25829.391,E2 25829.391} C_VEL
LIN {X 0,Y 559.91,Z 1281.086,A -85,B 0,C 180,E1 25827.241,E2 25827.241} C_VEL
LIN {X 0,Y 559.922,Z 1279.222,A -85,B 0,C 180,E1 25824.985,E2 25824.985} C_VEL
LIN {X 0,Y 559.965,Z 1276.222,A -85,B 0,C 180,E1 25822.722,E2 25822.722} C_VEL
LIN {X 0,Y 560.05,Z 1271.685,A -85,B 0,C 180,E1 25820.239,E2 25820.239} C_VEL
LIN {X 0,Y 560.377,Z 1264.579,A -85,B 0,C 180,E1 25817.328,E2 25817.328} C_VEL
LIN {X 0,Y 560.863,Z 1256.878,A -85,B 0,C 180,E1 25814.813,E2 25814.813} C_VEL
LIN {X 0,Y 561.462,Z 1248.915,A -85,B 0,C 180,E1 25812.597,E2 25812.597} C_VEL
LIN {X 0,Y 562.461,Z 1238.793,A -85,B 0,C 180,E1 25810.157,E2 25810.157} C_VEL
LIN {X 0,Y 563.983,Z 1225.322,A -85,B 0,C 180,E1 25807.38,E2 25807.38} C_VEL
LIN {X 0,Y 565.598,Z 1212.763,A -85,B 0,C 180,E1 25805.125,E2 25805.125} C_VEL
LIN {X 0,Y 567.448,Z 1199.997,A -85,B 0,C 180,E1 25803.077,E2 25803.077} C_VEL
LIN {X 0,Y 570.05,Z 1183.157,A -85,B 0,C 180,E1 25800.664,E2 25800.664} C_VEL
LIN {X 0,Y 572.949,Z 1165.271,A -85,B 0,C 180,E1 25798.437,E2 25798.437} C_VEL
LIN {X 0,Y 575.569,Z 1149.568,A -85,B 0,C 180,E1 25796.679,E2 25796.679} C_VEL
LIN {X 0,Y 578.44,Z 1132.779,A -85,B 0,C 180,E1 25794.986,E2 25794.986} C_VEL
LIN {X 0,Y 582.105,Z 1111.299,A -85,B 0,C 180,E1 25793.052,E2 25793.052} C_VEL
LIN {X 0,Y 585.61,Z 1090.055,A -85,B 0,C 180,E1 25791.395,E2 25791.395} C_VEL
LIN {X 0,Y 588.533,Z 1071.527,A -85,B 0,C 180,E1 25790.116,E2 25790.116} C_VEL
LIN {X 0,Y 591.537,Z 1051.666,A -85,B 0,C 180,E1 25788.897,E2 25788.897} C_VEL
LIN {X 0,Y 594.751,Z 1029.212,A -85,B 0,C 180,E1 25787.686,E2 25787.686} C_VEL
LIN {X 0,Y 598.144,Z 1002.818,A -85,B 0,C 180,E1 25786.48,E2 25786.48} C_VEL
LIN {X 0,Y 600.637,Z 981.126,A -85,B 0,C 180,E1 25785.648,E2 25785.648} C_VEL
LIN {X 0,Y 602.785,Z 959.868,A -85,B 0,C 180,E1 25784.958,E2 25784.958} C_VEL
LIN {X 0,Y 604.672,Z 938.512,A -85,B 0,C 180,E1 25784.389,E2 25784.389} C_VEL
LIN {X 0,Y 606.383,Z 914.746,A -85,B 0,C 180,E1 25783.886,E2 25783.886} C_VEL
LIN {X 0,Y 607.895,Z 878.562,A -85,B 0,C 180,E1 25783.33,E2 25783.33} C_VEL
LIN {X 0,Y 614.516,Z 654.204,A -85,B 0,C 180,E1 25780.158,E2 25780.158} C_VEL
LIN {X 0,Y 619.457,Z 494.927,A -85,B 0,C 180,E1 25777.849,E2 25777.849} C_VEL
LIN {X 0,Y 606.65,Z 475.537,A -85,B 0,C 180,E1 25775.899,E2 25775.899} C_VEL
LIN {X 0,Y 596.292,Z 460.72,A -85,B 0,C 180,E1 25774.206,E2 25774.206} C_VEL
LIN {X 0,Y 585.758,Z 446.306,A -85,B 0,C 180,E1 25772.354,E2 25772.354} C_VEL
LIN {X 0,Y 582.116,Z 441.54,A -85,B 0,C 180,E1 25771.681,E2 25771.681} C_VEL
LIN {X 0,Y 577.644,Z 435.617,A -85,B 0,C 180,E1 25770.822,E2 25770.822} C_VEL
LIN {X 0,Y 570.306,Z 426.253,A -85,B 0,C 180,E1 25769.343,E2 25769.343} C_VEL
LIN {X 0,Y 567.093,Z 422.044,A -85,B 0,C 180,E1 25768.659,E2 25768.659} C_VEL
LIN {X 0,Y 565.608,Z 419.91,A -85,B 0,C 180,E1 25768.165,E2 25768.165} C_VEL
LIN {X 0,Y 563.849,Z 416.128,A -85,B 0,C 180,E1 25767.339,E2 25767.339} C_VEL
LIN {X 0,Y 561.812,Z 413.078,A -85,B 0,C 180,E1 25766.534,E2 25766.534} C_VEL
LIN {X 0,Y 561.394,Z 411.26,A -85,B 0,C 180,E1 25766.165,E2 25766.165} C_VEL
LIN {X 0,Y 561.367,Z 411.307,A -85,B 0,C 180,E1 25762.849,E2 25762.849} C_VEL
LIN {X 0,Y 561.408,Z 411.249,A -85,B 0,C 180,E1 25759.779,E2 25759.779} C_VEL
LIN {X 0,Y 561.351,Z 411.284,A -85,B 0,C 180,E1 25756.559,E2 25756.559} C_VEL
LIN {X 0,Y 561.421,Z 411.265,A -85,B 0,C 180,E1 25753.387,E2 25753.387} C_VEL
LIN {X 0,Y 561.336,Z 411.267,A -85,B 0,C 180,E1 25750.261,E2 25750.261} C_VEL
LIN {X 0,Y 561.395,Z 411.285,A -85,B 0,C 180,E1 25747.059,E2 25747.059} C_VEL
LIN {X 0,Y 561.339,Z 411.26,A -85,B 0,C 180,E1 25743.983,E2 25743.983} C_VEL
LIN {X 0,Y 561.383,Z 411.295,A -85,B 0,C 180,E1 25740.714,E2 25740.714} C_VEL
LIN {X 0,Y 561.351,Z 411.256,A -85,B 0,C 180,E1 25737.754,E2 25737.754} C_VEL
LIN {X 0,Y 561.379,Z 411.304,A -85,B 0,C 180,E1 25734.378,E2 25734.378} C_VEL
LIN {X 0,Y 561.368,Z 411.252,A -85,B 0,C 180,E1 25731.498,E2 25731.498} C_VEL
LIN {X 0,Y 561.379,Z 411.303,A -85,B 0,C 180,E1 25728.076,E2 25728.076} C_VEL
LIN {X 0,Y 561.402,Z 411.246,A -85,B 0,C 180,E1 25725.033,E2 25725.033} C_VEL
LIN {X 0,Y 561.382,Z 411.299,A -85,B 0,C 180,E1 25721.731,E2 25721.731} C_VEL
LIN {X 0,Y 561.444,Z 411.252,A -85,B 0,C 180,E1 25718.477,E2 25718.477} C_VEL
LIN {X 0,Y 561.383,Z 411.264,A -85,B 0,C 180,E1 25715.368,E2 25715.368} C_VEL
LIN {X 0,Y 561.468,Z 411.452,A -85,B 0,C 180,E1 25712.177,E2 25712.177} C_VEL
LIN {X 0,Y 562.501,Z 414.425,A -85,B 0,C 180,E1 25711.897,E2 25711.897} C_VEL
LIN {X 0,Y 564.823,Z 416.907,A -85,B 0,C 180,E1 25711.389,E2 25711.389} C_VEL
LIN {X 0,Y 566.66,Z 418.158,A -85,B 0,C 180,E1 25711.015,E2 25711.015} C_VEL
LIN {X 0,Y 568.879,Z 421.75,A -85,B 0,C 180,E1 25710.518,E2 25710.518} C_VEL
LIN {X 0,Y 571.807,Z 424.463,A -85,B 0,C 180,E1 25709.931,E2 25709.931} C_VEL
LIN {X 0,Y 574.751,Z 428.496,A -85,B 0,C 180,E1 25709.325,E2 25709.325} C_VEL
LIN {X 0,Y 576.831,Z 430.507,A -85,B 0,C 180,E1 25708.927,E2 25708.927} C_VEL
LIN {X 0,Y 580.248,Z 434.918,A -85,B 0,C 180,E1 25708.263,E2 25708.263} C_VEL
LIN {X 0,Y 582.006,Z 436.925,A -85,B 0,C 180,E1 25707.936,E2 25707.936} C_VEL
LIN {X 0,Y 586.97,Z 443.115,A -85,B 0,C 180,E1 25707.026,E2 25707.026} C_VEL
LIN {X 0,Y 595.029,Z 453.174,A -85,B 0,C 180,E1 25705.624,E2 25705.624} C_VEL
LIN {X 0,Y 606.84,Z 468.658,A -85,B 0,C 180,E1 25703.705,E2 25703.705} C_VEL
LIN {X 0,Y 619.331,Z 485.955,A -85,B 0,C 180,E1 25701.825,E2 25701.825} C_VEL
LIN {X 0,Y 612.321,Z 707.035,A -85,B 0,C 180,E1 25698.645,E2 25698.645} C_VEL
LIN {X 0,Y 610.089,Z 781.231,A -85,B 0,C 180,E1 25697.594,E2 25697.594} C_VEL
LIN {X 0,Y 609.189,Z 788.935,A -85,B 0,C 180,E1 25697.555,E2 25697.555} C_VEL
LIN {X 0,Y 604.359,Z 809.57,A -85,B 0,C 180,E1 25697.703,E2 25697.703} C_VEL
LIN {X 0,Y 603.651,Z 816.179,A -85,B 0,C 180,E1 25697.663,E2 25697.663} C_VEL
LIN {X 0,Y 601.544,Z 878.005,A -85,B 0,C 180,E1 25696.767,E2 25696.767} C_VEL
LIN {X 0,Y 599.611,Z 906.947,A -85,B 0,C 180,E1 25696.197,E2 25696.197} C_VEL
LIN {X 0,Y 597.505,Z 930.401,A -85,B 0,C 180,E1 25695.576,E2 25695.576} C_VEL
LIN {X 0,Y 595.375,Z 950.741,A -85,B 0,C 180,E1 25694.917,E2 25694.917} C_VEL
LIN {X 0,Y 592.91,Z 971.197,A -85,B 0,C 180,E1 25694.136,E2 25694.136} C_VEL
LIN {X 0,Y 590.119,Z 992.365,A -85,B 0,C 180,E1 25693.19,E2 25693.19} C_VEL
LIN {X 0,Y 586.384,Z 1017.597,A -85,B 0,C 180,E1 25691.871,E2 25691.871} C_VEL
LIN {X 0,Y 582.801,Z 1039.41,A -85,B 0,C 180,E1 25690.532,E2 25690.532} C_VEL
LIN {X 0,Y 579.675,Z 1057.619,A -85,B 0,C 180,E1 25689.266,E2 25689.266} C_VEL
LIN {X 0,Y 576.725,Z 1074.239,A -85,B 0,C 180,E1 25687.978,E2 25687.978} C_VEL
LIN {X 0,Y 573.129,Z 1094.313,A -85,B 0,C 180,E1 25686.25,E2 25686.25} C_VEL
LIN {X 0,Y 569.135,Z 1116.431,A -85,B 0,C 180,E1 25684.078,E2 25684.078} C_VEL
LIN {X 0,Y 566.178,Z 1133.07,A -85,B 0,C 180,E1 25682.224,E2 25682.224} C_VEL
LIN {X 0,Y 563.566,Z 1148.084,A -85,B 0,C 180,E1 25680.367,E2 25680.367} C_VEL
LIN {X 0,Y 560.782,Z 1164.952,A -85,B 0,C 180,E1 25678.042,E2 25678.042} C_VEL
LIN {X 0,Y 558.287,Z 1181.024,A -85,B 0,C 180,E1 25675.489,E2 25675.489} C_VEL
LIN {X 0,Y 556.548,Z 1193.369,A -85,B 0,C 180,E1 25673.275,E2 25673.275} C_VEL
LIN {X 0,Y 555.06,Z 1205.172,A -85,B 0,C 180,E1 25670.89,E2 25670.89} C_VEL
LIN {X 0,Y 553.739,Z 1217.532,A -85,B 0,C 180,E1 25667.979,E2 25667.979} C_VEL
LIN {X 0,Y 552.991,Z 1226.023,A -85,B 0,C 180,E1 25665.624,E2 25665.624} C_VEL
LIN {X 0,Y 552.513,Z 1232.935,A -85,B 0,C 180,E1 25663.388,E2 25663.388} C_VEL
LIN {X 0,Y 552.202,Z 1238.722,A -85,B 0,C 180,E1 25661.166,E2 25661.166} C_VEL
LIN {X 0,Y 552.026,Z 1244.075,A -85,B 0,C 180,E1 25658.641,E2 25658.641} C_VEL
LIN {X 0,Y 551.935,Z 1248.488,A -85,B 0,C 180,E1 25655.713,E2 25655.713} C_VEL
LIN {X 0,Y 551.911,Z 1250.716,A -85,B 0,C 180,E1 25653.319,E2 25653.319} C_VEL
LIN {X 0,Y 551.888,Z 1251.75,A -85,B 0,C 180,E1 25651.137,E2 25651.137} C_VEL
LIN {X 0,Y 551.869,Z 1251.813,A -85,B 0,C 180,E1 25649.061,E2 25649.061} C_VEL
LIN {X 0,Y 551.909,Z 1250.973,A -85,B 0,C 180,E1 25646.984,E2 25646.984} C_VEL
LIN {X 0,Y 551.923,Z 1249.031,A -85,B 0,C 180,E1 25644.694,E2 25644.694} C_VEL
LIN {X 0,Y 551.958,Z 1245.795,A -85,B 0,C 180,E1 25642.292,E2 25642.292} C_VEL
LIN {X 0,Y 552.149,Z 1240.597,A -85,B 0,C 180,E1 25639.523,E2 25639.523} C_VEL
LIN {X 0,Y 552.476,Z 1233.77,A -85,B 0,C 180,E1 25636.814,E2 25636.814} C_VEL
LIN {X 0,Y 552.945,Z 1226.642,A -85,B 0,C 180,E1 25634.473,E2 25634.473} C_VEL
LIN {X 0,Y 553.626,Z 1218.64,A -85,B 0,C 180,E1 25632.224,E2 25632.224} C_VEL
LIN {X 0,Y 554.756,Z 1208.007,A -85,B 0,C 180,E1 25629.64,E2 25629.64} C_VEL
LIN {X 0,Y 556.339,Z 1194.919,A -85,B 0,C 180,E1 25626.93,E2 25626.93} C_VEL
LIN {X 0,Y 557.987,Z 1182.952,A -85,B 0,C 180,E1 25624.752,E2 25624.752} C_VEL
LIN {X 0,Y 559.926,Z 1170.221,A -85,B 0,C 180,E1 25622.678,E2 25622.678} C_VEL
LIN {X 0,Y 562.652,Z 1153.692,A -85,B 0,C 180,E1 25620.273,E2 25620.273} C_VEL
LIN {X 0,Y 565.798,Z 1135.301,A -85,B 0,C 180,E1 25617.95,E2 25617.95} C_VEL
LIN {X 0,Y 568.561,Z 1119.623,A -85,B 0,C 180,E1 25616.175,E2 25616.175} C_VEL
LIN {X 0,Y 571.536,Z 1103.083,A -85,B 0,C 180,E1 25614.488,E2 25614.488} C_VEL
LIN {X 0,Y 575.407,Z 1081.669,A -85,B 0,C 180,E1 25612.538,E2 25612.538} C_VEL
LIN {X 0,Y 579.133,Z 1060.703,A -85,B 0,C 180,E1 25610.87,E2 25610.87} C_VEL
LIN {X 0,Y 582.392,Z 1041.765,A -85,B 0,C 180,E1 25609.533,E2 25609.533} C_VEL
LIN {X 0,Y 585.445,Z 1023.118,A -85,B 0,C 180,E1 25608.362,E2 25608.362} C_VEL
LIN {X 0,Y 588.684,Z 1002.087,A -85,B 0,C 180,E1 25607.2,E2 25607.2} C_VEL
LIN {X 0,Y 592.42,Z 975.222,A -85,B 0,C 180,E1 25605.94,E2 25605.94} C_VEL
LIN {X 0,Y 595.101,Z 953.156,A -85,B 0,C 180,E1 25605.078,E2 25605.078} C_VEL
LIN {X 0,Y 597.319,Z 932.249,A -85,B 0,C 180,E1 25604.389,E2 25604.389} C_VEL
LIN {X 0,Y 599.265,Z 911.036,A -85,B 0,C 180,E1 25603.814,E2 25603.814} C_VEL
LIN {X 0,Y 600.966,Z 887.962,A -85,B 0,C 180,E1 25603.316,E2 25603.316} C_VEL
LIN {X 0,Y 602.559,Z 852.192,A -85,B 0,C 180,E1 25602.757,E2 25602.757} C_VEL
LIN {X 0,Y 609.568,Z 630.089,A -85,B 0,C 180,E1 25599.588,E2 25599.588} C_VEL
LIN {X 0,Y 614.19,Z 490.048,A -85,B 0,C 180,E1 25597.54,E2 25597.54} C_VEL
LIN {X 0,Y 601.785,Z 472.849,A -85,B 0,C 180,E1 25595.618,E2 25595.618} C_VEL
LIN {X 0,Y 590.541,Z 458.076,A -85,B 0,C 180,E1 25593.736,E2 25593.736} C_VEL
LIN {X 0,Y 581.917,Z 447.258,A -85,B 0,C 180,E1 25592.186,E2 25592.186} C_VEL
LIN {X 0,Y 577.625,Z 441.975,A -85,B 0,C 180,E1 25591.373,E2 25591.373} C_VEL
LIN {X 0,Y 573.101,Z 436.426,A -85,B 0,C 180,E1 25590.482,E2 25590.482} C_VEL
LIN {X 0,Y 569.565,Z 432.164,A -85,B 0,C 180,E1 25589.761,E2 25589.761} C_VEL
LIN {X 0,Y 568.369,Z 430.708,A -85,B 0,C 180,E1 25589.511,E2 25589.511} C_VEL
LIN {X 0,Y 565.111,Z 427.22,A -85,B 0,C 180,E1 25588.826,E2 25588.826} C_VEL
LIN {X 0,Y 563.687,Z 424.962,A -85,B 0,C 180,E1 25588.5,E2 25588.5} C_VEL
LIN {X 0,Y 560.58,Z 422.267,A -85,B 0,C 180,E1 25587.832,E2 25587.832} C_VEL
LIN {X 0,Y 558.549,Z 418.746,A -85,B 0,C 180,E1 25587.334,E2 25587.334} C_VEL
LIN {X 0,Y 555.413,Z 416.531,A -85,B 0,C 180,E1 25586.633,E2 25586.633} C_VEL
LIN {X 0,Y 553.797,Z 413.655,A -85,B 0,C 180,E1 25586.211,E2 25586.211} C_VEL
LIN {X 0,Y 553.49,Z 412.236,A -85,B 0,C 180,E1 25586.103,E2 25586.103} C_VEL
LIN {X 0,Y 553.504,Z 412.281,A -85,B 0,C 180,E1 25582.611,E2 25582.611} C_VEL
LIN {X 0,Y 553.479,Z 412.246,A -85,B 0,C 180,E1 25579.196,E2 25579.196} C_VEL
LIN {X 0,Y 553.489,Z 412.243,A -85,B 0,C 180,E1 25575.938,E2 25575.938} C_VEL
LIN {X 0,Y 553.485,Z 412.275,A -85,B 0,C 180,E1 25572.626,E2 25572.626} C_VEL
LIN {X 0,Y 553.49,Z 412.227,A -85,B 0,C 180,E1 25569.252,E2 25569.252} C_VEL
LIN {X 0,Y 553.502,Z 412.288,A -85,B 0,C 180,E1 25565.91,E2 25565.91} C_VEL
LIN {X 0,Y 553.47,Z 412.226,A -85,B 0,C 180,E1 25562.485,E2 25562.485} C_VEL
LIN {X 0,Y 553.5,Z 412.28,A -85,B 0,C 180,E1 25559.172,E2 25559.172} C_VEL
LIN {X 0,Y 553.487,Z 412.232,A -85,B 0,C 180,E1 25555.732,E2 25555.732} C_VEL
LIN {X 0,Y 553.479,Z 412.257,A -85,B 0,C 180,E1 25552.422,E2 25552.422} C_VEL
LIN {X 0,Y 553.496,Z 412.253,A -85,B 0,C 180,E1 25549.066,E2 25549.066} C_VEL
LIN {X 0,Y 553.469,Z 412.238,A -85,B 0,C 180,E1 25545.777,E2 25545.777} C_VEL
LIN {X 0,Y 553.501,Z 412.285,A -85,B 0,C 180,E1 25542.441,E2 25542.441} C_VEL
LIN {X 0,Y 553.494,Z 412.236,A -85,B 0,C 180,E1 25539.042,E2 25539.042} C_VEL
LIN {X 0,Y 553.47,Z 412.248,A -85,B 0,C 180,E1 25535.789,E2 25535.789} C_VEL
LIN {X 0,Y 553.487,Z 412.38,A -85,B 0,C 180,E1 25535.284,E2 25535.284} C_VEL
LIN {X 0,Y 554.86,Z 415.804,A -85,B 0,C 180,E1 25534.488,E2 25534.488} C_VEL
LIN {X 0,Y 556.392,Z 417.883,A -85,B 0,C 180,E1 25533.878,E2 25533.878} C_VEL
LIN {X 0,Y 558.193,Z 421.453,A -85,B 0,C 180,E1 25533.08,E2 25533.08} C_VEL
LIN {X 0,Y 560.128,Z 423.717,A -85,B 0,C 180,E1 25532.634,E2 25532.634} C_VEL
LIN {X 0,Y 563.53,Z 427.896,A -85,B 0,C 180,E1 25531.869,E2 25531.869} C_VEL
LIN {X 0,Y 565.313,Z 430.291,A -85,B 0,C 180,E1 25531.474,E2 25531.474} C_VEL
LIN {X 0,Y 570.164,Z 436.416,A -85,B 0,C 180,E1 25530.444,E2 25530.444} C_VEL
LIN {X 0,Y 577.513,Z 445.98,A -85,B 0,C 180,E1 25528.968,E2 25528.968} C_VEL
LIN {X 0,Y 585.778,Z 456.965,A -85,B 0,C 180,E1 25527.415,E2 25527.415} C_VEL
LIN {X 0,Y 596.454,Z 472.019,A -85,B 0,C 180,E1 25525.543,E2 25525.543} C_VEL
LIN {X 0,Y 608.128,Z 489.215,A -85,B 0,C 180,E1 25523.648,E2 25523.648} C_VEL
LIN {X 0,Y 614.477,Z 499.433,A -85,B 0,C 180,E1 25522.665,E2 25522.665} C_VEL
LIN {X 0,Y 607.221,Z 720.611,A -85,B 0,C 180,E1 25519.466,E2 25519.466} C_VEL
LIN {X 0,Y 601.492,Z 902.32,A -85,B 0,C 180,E1 25516.872,E2 25516.872} C_VEL
LIN {X 0,Y 599.984,Z 926.542,A -85,B 0,C 180,E1 25516.432,E2 25516.432} C_VEL
LIN {X 0,Y 597.538,Z 955.158,A -85,B 0,C 180,E1 25515.722,E2 25515.722} C_VEL
LIN {X 0,Y 595.277,Z 976.863,A -85,B 0,C 180,E1 25515.041,E2 25515.041} C_VEL
LIN {X 0,Y 592.886,Z 997.139,A -85,B 0,C 180,E1 25514.286,E2 25514.286} C_VEL
LIN {X 0,Y 590.39,Z 1016.579,A -85,B 0,C 180,E1 25513.444,E2 25513.444} C_VEL
LIN {X 0,Y 587.509,Z 1036.855,A -85,B 0,C 180,E1 25512.442,E2 25512.442} C_VEL
LIN {X 0,Y 583.863,Z 1061.223,A -85,B 0,C 180,E1 25511.056,E2 25511.056} C_VEL
LIN {X 0,Y 580.025,Z 1084.485,A -85,B 0,C 180,E1 25509.505,E2 25509.505} C_VEL
LIN {X 0,Y 576.848,Z 1103.162,A -85,B 0,C 180,E1 25508.098,E2 25508.098} C_VEL
LIN {X 0,Y 574.028,Z 1119.227,A -85,B 0,C 180,E1 25506.748,E2 25506.748} C_VEL
LIN {X 0,Y 571.12,Z 1135.452,A -85,B 0,C 180,E1 25505.234,E2 25505.234} C_VEL
LIN {X 0,Y 568.183,Z 1151.78,A -85,B 0,C 180,E1 25503.547,E2 25503.547} C_VEL
LIN {X 0,Y 564.881,Z 1170.712,A -85,B 0,C 180,E1 25501.363,E2 25501.363} C_VEL
LIN {X 0,Y 561.897,Z 1188.035,A -85,B 0,C 180,E1 25499.068,E2 25499.068} C_VEL
LIN {X 0,Y 559.759,Z 1201.348,A -85,B 0,C 180,E1 25497.101,E2 25497.101} C_VEL
LIN {X 0,Y 557.742,Z 1214.605,A -85,B 0,C 180,E1 25494.92,E2 25494.92} C_VEL
LIN {X 0,Y 555.787,Z 1229.142,A -85,B 0,C 180,E1 25492.201,E2 25492.201} C_VEL
LIN {X 0,Y 554.445,Z 1240.587,A -85,B 0,C 180,E1 25489.712,E2 25489.712} C_VEL
LIN {X 0,Y 553.513,Z 1249.687,A -85,B 0,C 180,E1 25487.454,E2 25487.454} C_VEL
LIN {X 0,Y 552.866,Z 1257.907,A -85,B 0,C 180,E1 25485.1,E2 25485.1} C_VEL
LIN {X 0,Y 552.313,Z 1266.514,A -85,B 0,C 180,E1 25482.127,E2 25482.127} C_VEL
LIN {X 0,Y 552.046,Z 1272.079,A -85,B 0,C 180,E1 25479.702,E2 25479.702} C_VEL
LIN {X 0,Y 551.96,Z 1276.206,A -85,B 0,C 180,E1 25477.394,E2 25477.394} C_VEL
LIN {X 0,Y 551.923,Z 1279.209,A -85,B 0,C 180,E1 25475.097,E2 25475.097} C_VEL
LIN {X 0,Y 551.908,Z 1281.148,A -85,B 0,C 180,E1 25472.704,E2 25472.704} C_VEL
LIN {X 0,Y 551.894,Z 1281.985,A -85,B 0,C 180,E1 25469.901,E2 25469.901} C_VEL
LIN {X 0,Y 551.91,Z 1281.154,A -85,B 0,C 180,E1 25467.305,E2 25467.305} C_VEL
LIN {X 0,Y 551.922,Z 1279.219,A -85,B 0,C 180,E1 25464.912,E2 25464.912} C_VEL
LIN {X 0,Y 551.961,Z 1276.219,A -85,B 0,C 180,E1 25462.615,E2 25462.615} C_VEL
LIN {X 0,Y 552.063,Z 1271.809,A -85,B 0,C 180,E1 25460.161,E2 25460.161} C_VEL
LIN {X 0,Y 552.403,Z 1264.881,A -85,B 0,C 180,E1 25457.248,E2 25457.248} C_VEL
LIN {X 0,Y 552.912,Z 1257.231,A -85,B 0,C 180,E1 25454.697,E2 25454.697} C_VEL
LIN {X 0,Y 553.551,Z 1249.319,A -85,B 0,C 180,E1 25452.449,E2 25452.449} C_VEL
LIN {X 0,Y 554.548,Z 1239.716,A -85,B 0,C 180,E1 25450.082,E2 25450.082} C_VEL
LIN {X 0,Y 556.144,Z 1226.466,A -85,B 0,C 180,E1 25447.267,E2 25447.267} C_VEL
LIN {X 0,Y 557.92,Z 1213.396,A -85,B 0,C 180,E1 25444.872,E2 25444.872} C_VEL
LIN {X 0,Y 559.854,Z 1200.712,A -85,B 0,C 180,E1 25442.8,E2 25442.8} C_VEL
LIN {X 0,Y 562.407,Z 1185.023,A -85,B 0,C 180,E1 25440.504,E2 25440.504} C_VEL
LIN {X 0,Y 565.649,Z 1166.195,A -85,B 0,C 180,E1 25438.101,E2 25438.101} C_VEL
LIN {X 0,Y 568.416,Z 1150.455,A -85,B 0,C 180,E1 25436.31,E2 25436.31} C_VEL
LIN {X 0,Y 571.345,Z 1134.171,A -85,B 0,C 180,E1 25434.64,E2 25434.64} C_VEL
LIN {X 0,Y 574.555,Z 1116.237,A -85,B 0,C 180,E1 25432.985,E2 25432.985} C_VEL
LIN {X 0,Y 578.495,Z 1093.522,A -85,B 0,C 180,E1 25431.148,E2 25431.148} C_VEL
LIN {X 0,Y 582.039,Z 1072.073,A -85,B 0,C 180,E1 25429.644,E2 25429.644} C_VEL
LIN {X 0,Y 585.174,Z 1052.302,A -85,B 0,C 180,E1 25428.416,E2 25428.416} C_VEL
LIN {X 0,Y 588.318,Z 1031.283,A -85,B 0,C 180,E1 25427.266,E2 25427.266} C_VEL
LIN {X 0,Y 592.072,Z 1003.844,A -85,B 0,C 180,E1 25425.987,E2 25425.987} C_VEL
LIN {X 0,Y 594.833,Z 980.858,A -85,B 0,C 180,E1 25425.099,E2 25425.099} C_VEL
LIN {X 0,Y 597.069,Z 959.684,A -85,B 0,C 180,E1 25424.409,E2 25424.409} C_VEL
LIN {X 0,Y 599.025,Z 938.387,A -85,B 0,C 180,E1 25423.839,E2 25423.839} C_VEL
LIN {X 0,Y 600.811,Z 914.645,A -85,B 0,C 180,E1 25423.335,E2 25423.335} C_VEL
LIN {X 0,Y 602.39,Z 878.528,A -85,B 0,C 180,E1 25422.776,E2 25422.776} C_VEL
LIN {X 0,Y 609.343,Z 654.052,A -85,B 0,C 180,E1 25419.58,E2 25419.58} C_VEL
LIN {X 0,Y 614.381,Z 499.029,A -85,B 0,C 180,E1 25417.318,E2 25417.318} C_VEL
LIN {X 0,Y 603.093,Z 481.749,A -85,B 0,C 180,E1 25415.558,E2 25415.558} C_VEL
LIN {X 0,Y 592.477,Z 466.412,A -85,B 0,C 180,E1 25413.785,E2 25413.785} C_VEL
LIN {X 0,Y 580.346,Z 449.631,A -85,B 0,C 180,E1 25411.585,E2 25411.585} C_VEL
LIN {X 0,Y 571.851,Z 438.618,A -85,B 0,C 180,E1 25409.918,E2 25409.918} C_VEL
LIN {X 0,Y 567.488,Z 433.06,A -85,B 0,C 180,E1 25409.011,E2 25409.011} C_VEL
LIN {X 0,Y 563.382,Z 427.787,A -85,B 0,C 180,E1 25408.119,E2 25408.119} C_VEL
LIN {X 0,Y 560.057,Z 423.616,A -85,B 0,C 180,E1 25407.369,E2 25407.369} C_VEL
LIN {X 0,Y 557.273,Z 420.25,A -85,B 0,C 180,E1 25406.652,E2 25406.652} C_VEL
LIN {X 0,Y 555.879,Z 417.026,A -85,B 0,C 180,E1 25405.919,E2 25405.919} C_VEL
LIN {X 0,Y 553.75,Z 413.695,A -85,B 0,C 180,E1 25404.994,E2 25404.994} C_VEL
LIN {X 0,Y 553.421,Z 412.245,A -85,B 0,C 180,E1 25404.668,E2 25404.668} C_VEL
LIN {X 0,Y 553.487,Z 412.25,A -85,B 0,C 180,E1 25401.514,E2 25401.514} C_VEL
LIN {X 0,Y 553.42,Z 412.277,A -85,B 0,C 180,E1 25398.323,E2 25398.323} C_VEL
LIN {X 0,Y 553.429,Z 412.237,A -85,B 0,C 180,E1 25394.973,E2 25394.973} C_VEL
LIN {X 0,Y 553.418,Z 412.295,A -85,B 0,C 180,E1 25391.992,E2 25391.992} C_VEL
LIN {X 0,Y 553.403,Z 412.241,A -85,B 0,C 180,E1 25388.625,E2 25388.625} C_VEL
LIN {X 0,Y 553.422,Z 412.293,A -85,B 0,C 180,E1 25385.703,E2 25385.703} C_VEL
LIN {X 0,Y 553.406,Z 412.243,A -85,B 0,C 180,E1 25382.382,E2 25382.382} C_VEL
LIN {X 0,Y 553.449,Z 412.282,A -85,B 0,C 180,E1 25379.379,E2 25379.379} C_VEL
LIN {X 0,Y 553.412,Z 412.245,A -85,B 0,C 180,E1 25376.063,E2 25376.063} C_VEL
LIN {X 0,Y 553.502,Z 412.264,A -85,B 0,C 180,E1 25372.84,E2 25372.84} C_VEL
LIN {X 0,Y 553.426,Z 412.254,A -85,B 0,C 180,E1 25369.591,E2 25369.591} C_VEL
LIN {X 0,Y 553.46,Z 412.249,A -85,B 0,C 180,E1 25366.31,E2 25366.31} C_VEL
LIN {X 0,Y 553.445,Z 412.267,A -85,B 0,C 180,E1 25363.306,E2 25363.306} C_VEL
LIN {X 0,Y 553.452,Z 412.236,A -85,B 0,C 180,E1 25359.924,E2 25359.924} C_VEL
LIN {X 0,Y 553.483,Z 412.289,A -85,B 0,C 180,E1 25356.807,E2 25356.807} C_VEL
LIN {X 0,Y 553.493,Z 412.47,A -85,B 0,C 180,E1 25353.774,E2 25353.774} C_VEL
LIN {X 0,Y 554.453,Z 415.248,A -85,B 0,C 180,E1 25353.491,E2 25353.491} C_VEL
LIN {X 0,Y 556.848,Z 417.847,A -85,B 0,C 180,E1 25352.923,E2 25352.923} C_VEL
LIN {X 0,Y 558.811,Z 419.122,A -85,B 0,C 180,E1 25352.492,E2 25352.492} C_VEL
LIN {X 0,Y 560.904,Z 422.708,A -85,B 0,C 180,E1 25351.983,E2 25351.983} C_VEL
LIN {X 0,Y 564.134,Z 425.51,A -85,B 0,C 180,E1 25351.293,E2 25351.293} C_VEL
LIN {X 0,Y 566.957,Z 429.471,A -85,B 0,C 180,E1 25350.67,E2 25350.67} C_VEL
LIN {X 0,Y 569.282,Z 431.769,A -85,B 0,C 180,E1 25350.194,E2 25350.194} C_VEL
LIN {X 0,Y 572.687,Z 436.081,A -85,B 0,C 180,E1 25349.493,E2 25349.493} C_VEL
LIN {X 0,Y 574.385,Z 437.974,A -85,B 0,C 180,E1 25349.158,E2 25349.158} C_VEL
LIN {X 0,Y 578.271,Z 442.613,A -85,B 0,C 180,E1 25348.404,E2 25348.404} C_VEL
LIN {X 0,Y 588.667,Z 455.738,A -85,B 0,C 180,E1 25346.493,E2 25346.493} C_VEL
LIN {X 0,Y 600.097,Z 470.592,A -85,B 0,C 180,E1 25344.56,E2 25344.56} C_VEL
LIN {X 0,Y 613.298,Z 488.722,A -85,B 0,C 180,E1 25342.502,E2 25342.502} C_VEL
LIN {X 0,Y 614.261,Z 490.538,A -85,B 0,C 180,E1 25342.35,E2 25342.35} C_VEL
LIN {X 0,Y 606.973,Z 710.148,A -85,B 0,C 180,E1 25339.172,E2 25339.172} C_VEL
LIN {X 0,Y 603.651,Z 816.179,A -85,B 0,C 180,E1 25337.663,E2 25337.663} C_VEL
LIN {X 0,Y 602.744,Z 823.881,A -85,B 0,C 180,E1 25337.624,E2 25337.624} C_VEL
LIN {X 0,Y 597.903,Z 844.511,A -85,B 0,C 180,E1 25337.776,E2 25337.776} C_VEL
LIN {X 0,Y 597.191,Z 851.118,A -85,B 0,C 180,E1 25337.735,E2 25337.735} C_VEL
LIN {X 0,Y 595.578,Z 887.18,A -85,B 0,C 180,E1 25337.174,E2 25337.174} C_VEL
LIN {X 0,Y 593.74,Z 911.154,A -85,B 0,C 180,E1 25336.658,E2 25336.658} C_VEL
LIN {X 0,Y 591.723,Z 932.412,A -85,B 0,C 180,E1 25336.08,E2 25336.08} C_VEL
LIN {X 0,Y 589.415,Z 953.376,A -85,B 0,C 180,E1 25335.387,E2 25335.387} C_VEL
LIN {X 0,Y 586.644,Z 975.304,A -85,B 0,C 180,E1 25334.527,E2 25334.527} C_VEL
LIN {X 0,Y 582.763,Z 1002.196,A -85,B 0,C 180,E1 25333.262,E2 25333.262} C_VEL
LIN {X 0,Y 579.375,Z 1023.298,A -85,B 0,C 180,E1 25332.089,E2 25332.089} C_VEL
LIN {X 0,Y 576.202,Z 1041.867,A -85,B 0,C 180,E1 25330.917,E2 25330.917} C_VEL
LIN {X 0,Y 572.926,Z 1060.078,A -85,B 0,C 180,E1 25329.625,E2 25329.625} C_VEL
LIN {X 0,Y 569.257,Z 1079.796,A -85,B 0,C 180,E1 25328.054,E2 25328.054} C_VEL
LIN {X 0,Y 564.911,Z 1102.125,A -85,B 0,C 180,E1 25326.012,E2 25326.012} C_VEL
LIN {X 0,Y 561.631,Z 1119.476,A -85,B 0,C 180,E1 25324.227,E2 25324.227} C_VEL
LIN {X 0,Y 558.707,Z 1135.174,A -85,B 0,C 180,E1 25322.432,E2 25322.432} C_VEL
LIN {X 0,Y 555.478,Z 1153.156,A -85,B 0,C 180,E1 25320.139,E2 25320.139} C_VEL
LIN {X 0,Y 552.539,Z 1169.74,A -85,B 0,C 180,E1 25317.708,E2 25317.708} C_VEL
LIN {X 0,Y 550.497,Z 1182.512,A -85,B 0,C 180,E1 25315.606,E2 25315.606} C_VEL
LIN {X 0,Y 548.643,Z 1195.101,A -85,B 0,C 180,E1 25313.287,E2 25313.287} C_VEL
LIN {X 0,Y 546.831,Z 1209.071,A -85,B 0,C 180,E1 25310.323,E2 25310.323} C_VEL
LIN {X 0,Y 545.749,Z 1218.748,A -85,B 0,C 180,E1 25307.921,E2 25307.921} C_VEL
LIN {X 0,Y 545.011,Z 1226.874,A -85,B 0,C 180,E1 25305.596,E2 25305.596} C_VEL
LIN {X 0,Y 544.499,Z 1234.148,A -85,B 0,C 180,E1 25303.156,E2 25303.156} C_VEL
LIN {X 0,Y 544.122,Z 1241.388,A -85,B 0,C 180,E1 25300.155,E2 25300.155} C_VEL
LIN {X 0,Y 543.956,Z 1245.989,A -85,B 0,C 180,E1 25297.6,E2 25297.6} C_VEL
LIN {X 0,Y 543.925,Z 1249.054,A -85,B 0,C 180,E1 25295.269,E2 25295.269} C_VEL
LIN {X 0,Y 543.91,Z 1250.989,A -85,B 0,C 180,E1 25292.946,E2 25292.946} C_VEL
LIN {X 0,Y 543.868,Z 1251.84,A -85,B 0,C 180,E1 25290.733,E2 25290.733} C_VEL
LIN {X 0,Y 543.907,Z 1251.676,A -85,B 0,C 180,E1 25288.415,E2 25288.415} C_VEL
LIN {X 0,Y 543.919,Z 1250.032,A -85,B 0,C 180,E1 25285.567,E2 25285.567} C_VEL
LIN {X 0,Y 543.961,Z 1246.909,A -85,B 0,C 180,E1 25282.921,E2 25282.921} C_VEL
LIN {X 0,Y 544.024,Z 1242.989,A -85,B 0,C 180,E1 25280.581,E2 25280.581} C_VEL
LIN {X 0,Y 544.26,Z 1238.15,A -85,B 0,C 180,E1 25278.337,E2 25278.337} C_VEL
LIN {X 0,Y 544.582,Z 1232.252,A -85,B 0,C 180,E1 25276.078,E2 25276.078} C_VEL
LIN {X 0,Y 545.215,Z 1224.517,A -85,B 0,C 180,E1 25273.591,E2 25273.591} C_VEL
LIN {X 0,Y 546.285,Z 1213.525,A -85,B 0,C 180,E1 25270.649,E2 25270.649} C_VEL
LIN {X 0,Y 547.489,Z 1203.474,A -85,B 0,C 180,E1 25268.347,E2 25268.347} C_VEL
LIN {X 0,Y 549.014,Z 1192.391,A -85,B 0,C 180,E1 25266.102,E2 25266.102} C_VEL
LIN {X 0,Y 551.136,Z 1178.496,A -85,B 0,C 180,E1 25263.606,E2 25263.606} C_VEL
LIN {X 0,Y 553.866,Z 1162.179,A -85,B 0,C 180,E1 25261.061,E2 25261.061} C_VEL
LIN {X 0,Y 556.47,Z 1147.234,A -85,B 0,C 180,E1 25258.992,E2 25258.992} C_VEL
LIN {X 0,Y 559.314,Z 1131.821,A -85,B 0,C 180,E1 25257.077,E2 25257.077} C_VEL
LIN {X 0,Y 563.113,Z 1111.957,A -85,B 0,C 180,E1 25254.875,E2 25254.875} C_VEL
LIN {X 0,Y 566.978,Z 1091.585,A -85,B 0,C 180,E1 25252.902,E2 25252.902} C_VEL
LIN {X 0,Y 570.15,Z 1074.995,A -85,B 0,C 180,E1 25251.46,E2 25251.46} C_VEL
LIN {X 0,Y 573.35,Z 1057.806,A -85,B 0,C 180,E1 25250.116,E2 25250.116} C_VEL
LIN {X 0,Y 576.616,Z 1039.612,A -85,B 0,C 180,E1 25248.843,E2 25248.843} C_VEL
LIN {X 0,Y 580.468,Z 1017.125,A -85,B 0,C 180,E1 25247.457,E2 25247.457} C_VEL
LIN {X 0,Y 584.199,Z 992.803,A -85,B 0,C 180,E1 25246.183,E2 25246.183} C_VEL
LIN {X 0,Y 587.09,Z 971.771,A -85,B 0,C 180,E1 25245.236,E2 25245.236} C_VEL
LIN {X 0,Y 589.64,Z 951.467,A -85,B 0,C 180,E1 25244.455,E2 25244.455} C_VEL
LIN {X 0,Y 591.93,Z 930.434,A -85,B 0,C 180,E1 25243.771,E2 25243.771} C_VEL
LIN {X 0,Y 594.187,Z 906.133,A -85,B 0,C 180,E1 25243.127,E2 25243.127} C_VEL
LIN {X 0,Y 596.109,Z 877.868,A -85,B 0,C 180,E1 25242.575,E2 25242.575} C_VEL
LIN {X 0,Y 598.481,Z 810.638,A -85,B 0,C 180,E1 25241.597,E2 25241.597} C_VEL
LIN {X 0,Y 605.78,Z 592.853,A -85,B 0,C 180,E1 25238.456,E2 25238.456} C_VEL
LIN {X 0,Y 609.24,Z 494.29,A -85,B 0,C 180,E1 25237.007,E2 25237.007} C_VEL
LIN {X 0,Y 595.769,Z 475.603,A -85,B 0,C 180,E1 25234.853,E2 25234.853} C_VEL
LIN {X 0,Y 583.536,Z 459.692,A -85,B 0,C 180,E1 25232.72,E2 25232.72} C_VEL
LIN {X 0,Y 574.839,Z 448.884,A -85,B 0,C 180,E1 25231.076,E2 25231.076} C_VEL
LIN {X 0,Y 570.245,Z 443.263,A -85,B 0,C 180,E1 25230.156,E2 25230.156} C_VEL
LIN {X 0,Y 566.553,Z 438.559,A -85,B 0,C 180,E1 25229.382,E2 25229.382} C_VEL
LIN {X 0,Y 562.464,Z 434.103,A -85,B 0,C 180,E1 25228.51,E2 25228.51} C_VEL
LIN {X 0,Y 561.03,Z 432.102,A -85,B 0,C 180,E1 25228.183,E2 25228.183} C_VEL
LIN {X 0,Y 557.689,Z 428.734,A -85,B 0,C 180,E1 25227.438,E2 25227.438} C_VEL
LIN {X 0,Y 555.94,Z 426.035,A -85,B 0,C 180,E1 25227.01,E2 25227.01} C_VEL
LIN {X 0,Y 552.692,Z 423.193,A -85,B 0,C 180,E1 25226.253,E2 25226.253} C_VEL
LIN {X 0,Y 550.683,Z 419.724,A -85,B 0,C 180,E1 25225.719,E2 25225.719} C_VEL
LIN {X 0,Y 547.525,Z 417.569,A -85,B 0,C 180,E1 25224.952,E2 25224.952} C_VEL
LIN {X 0,Y 545.881,Z 414.714,A -85,B 0,C 180,E1 25224.485,E2 25224.485} C_VEL
LIN {X 0,Y 545.55,Z 413.234,A -85,B 0,C 180,E1 25224.355,E2 25224.355} C_VEL
LIN {X 0,Y 545.541,Z 413.225,A -85,B 0,C 180,E1 25221.102,E2 25221.102} C_VEL
LIN {X 0,Y 545.562,Z 413.275,A -85,B 0,C 180,E1 25217.713,E2 25217.713} C_VEL
LIN {X 0,Y 545.557,Z 413.217,A -85,B 0,C 180,E1 25214.217,E2 25214.217} C_VEL
LIN {X 0,Y 545.541,Z 413.255,A -85,B 0,C 180,E1 25210.882,E2 25210.882} C_VEL
LIN {X 0,Y 545.557,Z 413.231,A -85,B 0,C 180,E1 25207.449,E2 25207.449} C_VEL
LIN {X 0,Y 545.548,Z 413.229,A -85,B 0,C 180,E1 25204.099,E2 25204.099} C_VEL
LIN {X 0,Y 545.539,Z 413.258,A -85,B 0,C 180,E1 25200.63,E2 25200.63} C_VEL
LIN {X 0,Y 545.552,Z 413.214,A -85,B 0,C 180,E1 25197.316,E2 25197.316} C_VEL
LIN {X 0,Y 545.543,Z 413.273,A -85,B 0,C 180,E1 25193.898,E2 25193.898} C_VEL
LIN {X 0,Y 545.537,Z 413.215,A -85,B 0,C 180,E1 25190.399,E2 25190.399} C_VEL
LIN {X 0,Y 545.56,Z 413.258,A -85,B 0,C 180,E1 25187.079,E2 25187.079} C_VEL
LIN {X 0,Y 545.528,Z 413.235,A -85,B 0,C 180,E1 25183.823,E2 25183.823} C_VEL
LIN {X 0,Y 545.559,Z 413.225,A -85,B 0,C 180,E1 25180.515,E2 25180.515} C_VEL
LIN {X 0,Y 545.55,Z 413.277,A -85,B 0,C 180,E1 25177.135,E2 25177.135} C_VEL
LIN {X 0,Y 545.568,Z 413.287,A -85,B 0,C 180,E1 25176.908,E2 25176.908} C_VEL
LIN {X 0,Y 546.88,Z 416.765,A -85,B 0,C 180,E1 25176.053,E2 25176.053} C_VEL
LIN {X 0,Y 548.564,Z 419.053,A -85,B 0,C 180,E1 25175.329,E2 25175.329} C_VEL
LIN {X 0,Y 549.605,Z 421.182,A -85,B 0,C 180,E1 25174.89,E2 25174.89} C_VEL
LIN {X 0,Y 553.069,Z 425.207,A -85,B 0,C 180,E1 25174.026,E2 25174.026} C_VEL
LIN {X 0,Y 557.827,Z 431.073,A -85,B 0,C 180,E1 25172.888,E2 25172.888} C_VEL
LIN {X 0,Y 562.452,Z 436.865,A -85,B 0,C 180,E1 25171.836,E2 25171.836} C_VEL
LIN {X 0,Y 568.086,Z 444.168,A -85,B 0,C 180,E1 25170.618,E2 25170.618} C_VEL
LIN {X 0,Y 574.721,Z 452.874,A -85,B 0,C 180,E1 25169.265,E2 25169.265} C_VEL
LIN {X 0,Y 583.373,Z 464.543,A -85,B 0,C 180,E1 25167.614,E2 25167.614} C_VEL
LIN {X 0,Y 595.098,Z 481.197,A -85,B 0,C 180,E1 25165.541,E2 25165.541} C_VEL
LIN {X 0,Y 607.893,Z 500.66,A -85,B 0,C 180,E1 25163.456,E2 25163.456} C_VEL
LIN {X 0,Y 609.462,Z 503.55,A -85,B 0,C 180,E1 25163.204,E2 25163.204} C_VEL
LIN {X 0,Y 601.808,Z 726.615,A -85,B 0,C 180,E1 25159.959,E2 25159.959} C_VEL
LIN {X 0,Y 596.02,Z 901.982,A -85,B 0,C 180,E1 25157.438,E2 25157.438} C_VEL
LIN {X 0,Y 594.458,Z 926.115,A -85,B 0,C 180,E1 25156.999,E2 25156.999} C_VEL
LIN {X 0,Y 591.901,Z 954.891,A -85,B 0,C 180,E1 25156.285,E2 25156.285} C_VEL
LIN {X 0,Y 589.458,Z 977.34,A -85,B 0,C 180,E1 25155.575,E2 25155.575} C_VEL
LIN {X 0,Y 586.886,Z 998.163,A -85,B 0,C 180,E1 25154.791,E2 25154.791} C_VEL
LIN {X 0,Y 584.128,Z 1018.6,A -85,B 0,C 180,E1 25153.891,E2 25153.891} C_VEL
LIN {X 0,Y 580.537,Z 1042.903,A -85,B 0,C 180,E1 25152.655,E2 25152.655} C_VEL
LIN {X 0,Y 576.611,Z 1066.741,A -85,B 0,C 180,E1 25151.223,E2 25151.223} C_VEL
LIN {X 0,Y 573.335,Z 1085.696,A -85,B 0,C 180,E1 25149.928,E2 25149.928} C_VEL
LIN {X 0,Y 570.175,Z 1103.396,A -85,B 0,C 180,E1 25148.578,E2 25148.578} C_VEL
LIN {X 0,Y 566.999,Z 1120.849,A -85,B 0,C 180,E1 25147.096,E2 25147.096} C_VEL
LIN {X 0,Y 563.99,Z 1137.116,A -85,B 0,C 180,E1 25145.56,E2 25145.56} C_VEL
LIN {X 0,Y 560.228,Z 1157.26,A -85,B 0,C 180,E1 25143.419,E2 25143.419} C_VEL
LIN {X 0,Y 556.728,Z 1175.793,A -85,B 0,C 180,E1 25141.151,E2 25141.151} C_VEL
LIN {X 0,Y 554.294,Z 1189.574,A -85,B 0,C 180,E1 25139.269,E2 25139.269} C_VEL
LIN {X 0,Y 551.955,Z 1203.447,A -85,B 0,C 180,E1 25137.166,E2 25137.166} C_VEL
LIN {X 0,Y 549.523,Z 1218.944,A -85,B 0,C 180,E1 25134.514,E2 25134.514} C_VEL
LIN {X 0,Y 547.701,Z 1231.803,A -85,B 0,C 180,E1 25131.964,E2 25131.964} C_VEL
LIN {X 0,Y 546.53,Z 1241.503,A -85,B 0,C 180,E1 25129.787,E2 25129.787} C_VEL
LIN {X 0,Y 545.523,Z 1250.901,A -85,B 0,C 180,E1 25127.387,E2 25127.387} C_VEL
LIN {X 0,Y 544.733,Z 1260.299,A -85,B 0,C 180,E1 25124.569,E2 25124.569} C_VEL
LIN {X 0,Y 544.296,Z 1267.535,A -85,B 0,C 180,E1 25121.877,E2 25121.877} C_VEL
LIN {X 0,Y 544.043,Z 1272.489,A -85,B 0,C 180,E1 25119.632,E2 25119.632} C_VEL
LIN {X 0,Y 543.961,Z 1276.362,A -85,B 0,C 180,E1 25117.397,E2 25117.397} C_VEL
LIN {X 0,Y 543.923,Z 1279.32,A -85,B 0,C 180,E1 25115.067,E2 25115.067} C_VEL
LIN {X 0,Y 543.907,Z 1281.283,A -85,B 0,C 180,E1 25112.533,E2 25112.533} C_VEL
LIN {X 0,Y 543.878,Z 1281.94,A -85,B 0,C 180,E1 25109.689,E2 25109.689} C_VEL
LIN {X 0,Y 543.91,Z 1281.086,A -85,B 0,C 180,E1 25107.16,E2 25107.16} C_VEL
LIN {X 0,Y 543.923,Z 1279.216,A -85,B 0,C 180,E1 25104.837,E2 25104.837} C_VEL
LIN {X 0,Y 543.958,Z 1276.216,A -85,B 0,C 180,E1 25102.506,E2 25102.506} C_VEL
LIN {X 0,Y 544.077,Z 1271.932,A -85,B 0,C 180,E1 25100.081,E2 25100.081} C_VEL
LIN {X 0,Y 544.431,Z 1265.184,A -85,B 0,C 180,E1 25097.166,E2 25097.166} C_VEL
LIN {X 0,Y 544.984,Z 1257.23,A -85,B 0,C 180,E1 25094.468,E2 25094.468} C_VEL
LIN {X 0,Y 545.689,Z 1249.318,A -85,B 0,C 180,E1 25092.188,E2 25092.188} C_VEL
LIN {X 0,Y 546.776,Z 1239.522,A -85,B 0,C 180,E1 25089.74,E2 25089.74} C_VEL
LIN {X 0,Y 548.533,Z 1225.891,A -85,B 0,C 180,E1 25086.82,E2 25086.82} C_VEL
LIN {X 0,Y 550.354,Z 1213.394,A -85,B 0,C 180,E1 25084.502,E2 25084.502} C_VEL
LIN {X 0,Y 552.382,Z 1200.71,A -85,B 0,C 180,E1 25082.401,E2 25082.401} C_VEL
LIN {X 0,Y 555.181,Z 1184.693,A -85,B 0,C 180,E1 25080.031,E2 25080.031} C_VEL
LIN {X 0,Y 558.528,Z 1166.194,A -85,B 0,C 180,E1 25077.645,E2 25077.645} C_VEL
LIN {X 0,Y 561.425,Z 1150.59,A -85,B 0,C 180,E1 25075.85,E2 25075.85} C_VEL
LIN {X 0,Y 564.473,Z 1134.45,A -85,B 0,C 180,E1 25074.175,E2 25074.175} C_VEL
LIN {X 0,Y 567.638,Z 1117.26,A -85,B 0,C 180,E1 25072.584,E2 25072.584} C_VEL
LIN {X 0,Y 571.755,Z 1094.733,A -85,B 0,C 180,E1 25070.732,E2 25070.732} C_VEL
LIN {X 0,Y 575.584,Z 1072.62,A -85,B 0,C 180,E1 25069.162,E2 25069.162} C_VEL
LIN {X 0,Y 578.853,Z 1052.939,A -85,B 0,C 180,E1 25067.925,E2 25067.925} C_VEL
LIN {X 0,Y 582.018,Z 1032.722,A -85,B 0,C 180,E1 25066.804,E2 25066.804} C_VEL
LIN {X 0,Y 585.554,Z 1008.55,A -85,B 0,C 180,E1 25065.642,E2 25065.642} C_VEL
LIN {X 0,Y 588.829,Z 982.822,A -85,B 0,C 180,E1 25064.618,E2 25064.618} C_VEL
LIN {X 0,Y 591.288,Z 960.664,A -85,B 0,C 180,E1 25063.885,E2 25063.885} C_VEL
LIN {X 0,Y 593.324,Z 939.572,A -85,B 0,C 180,E1 25063.311,E2 25063.311} C_VEL
LIN {X 0,Y 595.053,Z 917.8,A -85,B 0,C 180,E1 25062.837,E2 25062.837} C_VEL
LIN {X 0,Y 596.572,Z 890.421,A -85,B 0,C 180,E1 25062.381,E2 25062.381} C_VEL
LIN {X 0,Y 603.813,Z 666.153,A -85,B 0,C 180,E1 25059.169,E2 25059.169} C_VEL
LIN {X 0,Y 609.36,Z 503.115,A -85,B 0,C 180,E1 25056.778,E2 25056.778} C_VEL
LIN {X 0,Y 599.557,Z 487.957,A -85,B 0,C 180,E1 25055.212,E2 25055.212} C_VEL
LIN {X 0,Y 588.937,Z 472.443,A -85,B 0,C 180,E1 25053.402,E2 25053.402} C_VEL
LIN {X 0,Y 577.407,Z 456.382,A -85,B 0,C 180,E1 25051.27,E2 25051.27} C_VEL
LIN {X 0,Y 569.116,Z 445.502,A -85,B 0,C 180,E1 25049.613,E2 25049.613} C_VEL
LIN {X 0,Y 564.692,Z 439.843,A -85,B 0,C 180,E1 25048.676,E2 25048.676} C_VEL
LIN {X 0,Y 560.716,Z 434.715,A -85,B 0,C 180,E1 25047.796,E2 25047.796} C_VEL
LIN {X 0,Y 556.04,Z 428.898,A -85,B 0,C 180,E1 25046.715,E2 25046.715} C_VEL
LIN {X 0,Y 551.53,Z 423.396,A -85,B 0,C 180,E1 25045.619,E2 25045.619} C_VEL
LIN {X 0,Y 548.788,Z 419.919,A -85,B 0,C 180,E1 25044.877,E2 25044.877} C_VEL
LIN {X 0,Y 548.086,Z 418.205,A -85,B 0,C 180,E1 25044.464,E2 25044.464} C_VEL
LIN {X 0,Y 546.026,Z 415.154,A -85,B 0,C 180,E1 25043.529,E2 25043.529} C_VEL
LIN {X 0,Y 545.501,Z 413.274,A -85,B 0,C 180,E1 25043.072,E2 25043.072} C_VEL
LIN {X 0,Y 545.5,Z 413.225,A -85,B 0,C 180,E1 25040.046,E2 25040.046} C_VEL
LIN {X 0,Y 545.479,Z 413.263,A -85,B 0,C 180,E1 25036.726,E2 25036.726} C_VEL
LIN {X 0,Y 545.526,Z 413.236,A -85,B 0,C 180,E1 25033.569,E2 25033.569} C_VEL
LIN {X 0,Y 545.459,Z 413.242,A -85,B 0,C 180,E1 25030.349,E2 25030.349} C_VEL
LIN {X 0,Y 545.515,Z 413.262,A -85,B 0,C 180,E1 25027.054,E2 25027.054} C_VEL
LIN {X 0,Y 545.465,Z 413.23,A -85,B 0,C 180,E1 25023.889,E2 25023.889} C_VEL
LIN {X 0,Y 545.482,Z 413.284,A -85,B 0,C 180,E1 25020.42,E2 25020.42} C_VEL
LIN {X 0,Y 545.501,Z 413.221,A -85,B 0,C 180,E1 25017.374,E2 25017.374} C_VEL
LIN {X 0,Y 545.487,Z 413.283,A -85,B 0,C 180,E1 25014.108,E2 25014.108} C_VEL
LIN {X 0,Y 545.532,Z 413.216,A -85,B 0,C 180,E1 25011.032,E2 25011.032} C_VEL
LIN {X 0,Y 545.494,Z 413.283,A -85,B 0,C 180,E1 25007.724,E2 25007.724} C_VEL
LIN {X 0,Y 545.55,Z 413.219,A -85,B 0,C 180,E1 25004.479,E2 25004.479} C_VEL
LIN {X 0,Y 545.507,Z 413.255,A -85,B 0,C 180,E1 25001.291,E2 25001.291} C_VEL
LIN {X 0,Y 545.513,Z 413.251,A -85,B 0,C 180,E1 24997.816,E2 24997.816} C_VEL
LIN {X 0,Y 545.525,Z 413.381,A -85,B 0,C 180,E1 24995.52,E2 24995.52} C_VEL
LIN {X 0,Y 546.428,Z 416.086,A -85,B 0,C 180,E1 24995.226,E2 24995.226} C_VEL
LIN {X 0,Y 548.665,Z 418.617,A -85,B 0,C 180,E1 24994.642,E2 24994.642} C_VEL
LIN {X 0,Y 550.965,Z 420.099,A -85,B 0,C 180,E1 24994.093,E2 24994.093} C_VEL
LIN {X 0,Y 552.981,Z 423.617,A -85,B 0,C 180,E1 24993.56,E2 24993.56} C_VEL
LIN {X 0,Y 556.45,Z 426.668,A -85,B 0,C 180,E1 24992.757,E2 24992.757} C_VEL
LIN {X 0,Y 559.126,Z 430.533,A -85,B 0,C 180,E1 24992.118,E2 24992.118} C_VEL
LIN {X 0,Y 561.796,Z 433.007,A -85,B 0,C 180,E1 24991.537,E2 24991.537} C_VEL
LIN {X 0,Y 565.153,Z 437.256,A -85,B 0,C 180,E1 24990.799,E2 24990.799} C_VEL
LIN {X 0,Y 566.893,Z 439.192,A -85,B 0,C 180,E1 24990.434,E2 24990.434} C_VEL
LIN {X 0,Y 570.743,Z 443.756,A -85,B 0,C 180,E1 24989.64,E2 24989.64} C_VEL
LIN {X 0,Y 575.709,Z 449.764,A -85,B 0,C 180,E1 24988.656,E2 24988.656} C_VEL
LIN {X 0,Y 588.686,Z 466.315,A -85,B 0,C 180,E1 24986.261,E2 24986.261} C_VEL
LIN {X 0,Y 600.53,Z 482.179,A -85,B 0,C 180,E1 24984.267,E2 24984.267} C_VEL
LIN {X 0,Y 609.264,Z 494.545,A -85,B 0,C 180,E1 24982.892,E2 24982.892} C_VEL
LIN {X 0,Y 601.708,Z 712.212,A -85,B 0,C 180,E1 24979.723,E2 24979.723} C_VEL
LIN {X 0,Y 597.191,Z 851.118,A -85,B 0,C 180,E1 24977.735,E2 24977.735} C_VEL
LIN {X 0,Y 596.283,Z 858.827,A -85,B 0,C 180,E1 24977.699,E2 24977.699} C_VEL
LIN {X 0,Y 591.227,Z 879.418,A -85,B 0,C 180,E1 24977.84,E2 24977.84} C_VEL
LIN {X 0,Y 590.281,Z 885.968,A -85,B 0,C 180,E1 24977.774,E2 24977.774} C_VEL
LIN {X 0,Y 588.297,Z 911.024,A -85,B 0,C 180,E1 24977.237,E2 24977.237} C_VEL
LIN {X 0,Y 586.207,Z 932.373,A -85,B 0,C 180,E1 24976.656,E2 24976.656} C_VEL
LIN {X 0,Y 583.883,Z 952.778,A -85,B 0,C 180,E1 24975.982,E2 24975.982} C_VEL
LIN {X 0,Y 581.23,Z 973.036,A -85,B 0,C 180,E1 24975.194,E2 24975.194} C_VEL
LIN {X 0,Y 577.736,Z 997.412,A -85,B 0,C 180,E1 24974.077,E2 24974.077} C_VEL
LIN {X 0,Y 573.68,Z 1021.722,A -85,B 0,C 180,E1 24972.746,E2 24972.746} C_VEL
LIN {X 0,Y 570.32,Z 1040.621,A -85,B 0,C 180,E1 24971.558,E2 24971.558} C_VEL
LIN {X 0,Y 567.03,Z 1058.178,A -85,B 0,C 180,E1 24970.319,E2 24970.319} C_VEL
LIN {X 0,Y 563.659,Z 1075.458,A -85,B 0,C 180,E1 24968.957,E2 24968.957} C_VEL
LIN {X 0,Y 560.142,Z 1093.083,A -85,B 0,C 180,E1 24967.405,E2 24967.405} C_VEL
LIN {X 0,Y 555.849,Z 1114.254,A -85,B 0,C 180,E1 24965.298,E2 24965.298} C_VEL
LIN {X 0,Y 551.937,Z 1133.542,A -85,B 0,C 180,E1 24963.099,E2 24963.099} C_VEL
LIN {X 0,Y 549.114,Z 1148.092,A -85,B 0,C 180,E1 24961.255,E2 24961.255} C_VEL
LIN {X 0,Y 546.077,Z 1164.745,A -85,B 0,C 180,E1 24958.9,E2 24958.9} C_VEL
LIN {X 0,Y 543.258,Z 1180.648,A -85,B 0,C 180,E1 24956.318,E2 24956.318} C_VEL
LIN {X 0,Y 541.316,Z 1192.8,A -85,B 0,C 180,E1 24954.086,E2 24954.086} C_VEL
LIN {X 0,Y 539.724,Z 1203.652,A -85,B 0,C 180,E1 24951.851,E2 24951.851} C_VEL
LIN {X 0,Y 538.298,Z 1215.033,A -85,B 0,C 180,E1 24949.188,E2 24949.188} C_VEL
LIN {X 0,Y 537.238,Z 1225.32,A -85,B 0,C 180,E1 24946.316,E2 24946.316} C_VEL
LIN {X 0,Y 536.627,Z 1232.331,A -85,B 0,C 180,E1 24944.012,E2 24944.012} C_VEL
LIN {X 0,Y 536.302,Z 1238,A -85,B 0,C 180,E1 24941.812,E2 24941.812} C_VEL
LIN {X 0,Y 536.044,Z 1242.832,A -85,B 0,C 180,E1 24939.551,E2 24939.551} C_VEL
LIN {X 0,Y 535.971,Z 1246.786,A -85,B 0,C 180,E1 24937.175,E2 24937.175} C_VEL
LIN {X 0,Y 535.918,Z 1249.954,A -85,B 0,C 180,E1 24934.489,E2 24934.489} C_VEL
LIN {X 0,Y 535.907,Z 1251.659,A -85,B 0,C 180,E1 24931.599,E2 24931.599} C_VEL
LIN {X 0,Y 535.865,Z 1251.857,A -85,B 0,C 180,E1 24929.247,E2 24929.247} C_VEL
LIN {X 0,Y 535.909,Z 1251.04,A -85,B 0,C 180,E1 24927.001,E2 24927.001} C_VEL
LIN {X 0,Y 535.924,Z 1249.137,A -85,B 0,C 180,E1 24924.643,E2 24924.643} C_VEL
LIN {X 0,Y 535.962,Z 1246.107,A -85,B 0,C 180,E1 24922.276,E2 24922.276} C_VEL
LIN {X 0,Y 536.119,Z 1241.745,A -85,B 0,C 180,E1 24919.79,E2 24919.79} C_VEL
LIN {X 0,Y 536.514,Z 1234.674,A -85,B 0,C 180,E1 24916.744,E2 24916.744} C_VEL
LIN {X 0,Y 537.049,Z 1227.342,A -85,B 0,C 180,E1 24914.223,E2 24914.223} C_VEL
LIN {X 0,Y 537.821,Z 1219.442,A -85,B 0,C 180,E1 24911.908,E2 24911.908} C_VEL
LIN {X 0,Y 538.901,Z 1210.193,A -85,B 0,C 180,E1 24909.553,E2 24909.553} C_VEL
LIN {X 0,Y 540.601,Z 1197.772,A -85,B 0,C 180,E1 24906.795,E2 24906.795} C_VEL
LIN {X 0,Y 542.779,Z 1183.575,A -85,B 0,C 180,E1 24904.11,E2 24904.11} C_VEL
LIN {X 0,Y 544.931,Z 1170.771,A -85,B 0,C 180,E1 24901.956,E2 24901.956} C_VEL
LIN {X 0,Y 547.686,Z 1155.863,A -85,B 0,C 180,E1 24899.717,E2 24899.717} C_VEL
LIN {X 0,Y 551.391,Z 1136.444,A -85,B 0,C 180,E1 24897.163,E2 24897.163} C_VEL
LIN {X 0,Y 554.796,Z 1119.157,A -85,B 0,C 180,E1 24895.154,E2 24895.154} C_VEL
LIN {X 0,Y 558.312,Z 1101.974,A -85,B 0,C 180,E1 24893.354,E2 24893.354} C_VEL
LIN {X 0,Y 563.037,Z 1078.738,A -85,B 0,C 180,E1 24891.226,E2 24891.226} C_VEL
LIN {X 0,Y 566.591,Z 1060.498,A -85,B 0,C 180,E1 24889.764,E2 24889.764} C_VEL
LIN {X 0,Y 569.837,Z 1043.234,A -85,B 0,C 180,E1 24888.526,E2 24888.526} C_VEL
LIN {X 0,Y 573.175,Z 1024.524,A -85,B 0,C 180,E1 24887.331,E2 24887.331} C_VEL
LIN {X 0,Y 576.632,Z 1003.838,A -85,B 0,C 180,E1 24886.167,E2 24886.167} C_VEL
LIN {X 0,Y 580.603,Z 977.858,A -85,B 0,C 180,E1 24884.918,E2 24884.918} C_VEL
LIN {X 0,Y 583.691,Z 954.385,A -85,B 0,C 180,E1 24883.986,E2 24883.986} C_VEL
LIN {X 0,Y 586.126,Z 933.117,A -85,B 0,C 180,E1 24883.276,E2 24883.276} C_VEL
LIN {X 0,Y 588.206,Z 912.059,A -85,B 0,C 180,E1 24882.699,E2 24882.699} C_VEL
LIN {X 0,Y 589.998,Z 889.564,A -85,B 0,C 180,E1 24882.206,E2 24882.206} C_VEL
LIN {X 0,Y 591.697,Z 855.713,A -85,B 0,C 180,E1 24881.662,E2 24881.662} C_VEL
LIN {X 0,Y 599.381,Z 633.264,A -85,B 0,C 180,E1 24878.447,E2 24878.447} C_VEL
LIN {X 0,Y 604.212,Z 498.508,A -85,B 0,C 180,E1 24876.449,E2 24876.449} C_VEL
LIN {X 0,Y 592.056,Z 481.565,A -85,B 0,C 180,E1 24874.456,E2 24874.456} C_VEL
LIN {X 0,Y 580.469,Z 466.327,A -85,B 0,C 180,E1 24872.393,E2 24872.393} C_VEL
LIN {X 0,Y 571.841,Z 455.539,A -85,B 0,C 180,E1 24870.732,E2 24870.732} C_VEL
LIN {X 0,Y 567.41,Z 450.072,A -85,B 0,C 180,E1 24869.827,E2 24869.827} C_VEL
LIN {X 0,Y 562.992,Z 444.699,A -85,B 0,C 180,E1 24868.887,E2 24868.887} C_VEL
LIN {X 0,Y 559.333,Z 440.201,A -85,B 0,C 180,E1 24868.073,E2 24868.073} C_VEL
LIN {X 0,Y 554.924,Z 435.321,A -85,B 0,C 180,E1 24867.063,E2 24867.063} C_VEL
LIN {X 0,Y 553.569,Z 433.341,A -85,B 0,C 180,E1 24866.728,E2 24866.728} C_VEL
LIN {X 0,Y 550.186,Z 430.081,A -85,B 0,C 180,E1 24865.918,E2 24865.918} C_VEL
LIN {X 0,Y 548.562,Z 427.263,A -85,B 0,C 180,E1 24865.478,E2 24865.478} C_VEL
LIN {X 0,Y 545.271,Z 424.72,A -85,B 0,C 180,E1 24864.657,E2 24864.657} C_VEL
LIN {X 0,Y 543.257,Z 421.233,A -85,B 0,C 180,E1 24864.074,E2 24864.074} C_VEL
LIN {X 0,Y 542.278,Z 420.544,A -85,B 0,C 180,E1 24863.817,E2 24863.817} C_VEL
LIN {X 0,Y 539.371,Z 418.358,A -85,B 0,C 180,E1 24863.026,E2 24863.026} C_VEL
LIN {X 0,Y 537.855,Z 415.418,A -85,B 0,C 180,E1 24862.539,E2 24862.539} C_VEL
LIN {X 0,Y 537.616,Z 414.247,A -85,B 0,C 180,E1 24862.413,E2 24862.413} C_VEL
LIN {X 0,Y 537.602,Z 414.223,A -85,B 0,C 180,E1 24858.995,E2 24858.995} C_VEL
LIN {X 0,Y 537.619,Z 414.209,A -85,B 0,C 180,E1 24855.645,E2 24855.645} C_VEL
LIN {X 0,Y 537.621,Z 414.261,A -85,B 0,C 180,E1 24852.132,E2 24852.132} C_VEL
LIN {X 0,Y 537.594,Z 414.201,A -85,B 0,C 180,E1 24848.773,E2 24848.773} C_VEL
LIN {X 0,Y 537.621,Z 414.26,A -85,B 0,C 180,E1 24845.443,E2 24845.443} C_VEL
LIN {X 0,Y 537.607,Z 414.202,A -85,B 0,C 180,E1 24842.025,E2 24842.025} C_VEL
LIN {X 0,Y 537.602,Z 414.237,A -85,B 0,C 180,E1 24838.615,E2 24838.615} C_VEL
LIN {X 0,Y 537.615,Z 414.217,A -85,B 0,C 180,E1 24835.199,E2 24835.199} C_VEL
LIN {X 0,Y 537.597,Z 414.214,A -85,B 0,C 180,E1 24831.874,E2 24831.874} C_VEL
LIN {X 0,Y 537.608,Z 414.252,A -85,B 0,C 180,E1 24828.412,E2 24828.412} C_VEL
LIN {X 0,Y 537.619,Z 414.203,A -85,B 0,C 180,E1 24825.018,E2 24825.018} C_VEL
LIN {X 0,Y 537.593,Z 414.248,A -85,B 0,C 180,E1 24821.68,E2 24821.68} C_VEL
LIN {X 0,Y 537.628,Z 414.275,A -85,B 0,C 180,E1 24818.685,E2 24818.685} C_VEL
LIN {X 0,Y 538.907,Z 417.748,A -85,B 0,C 180,E1 24817.759,E2 24817.759} C_VEL
LIN {X 0,Y 540.797,Z 419.985,A -85,B 0,C 180,E1 24816.98,E2 24816.98} C_VEL
LIN {X 0,Y 543.74,Z 424.13,A -85,B 0,C 180,E1 24816.136,E2 24816.136} C_VEL
LIN {X 0,Y 546.083,Z 426.559,A -85,B 0,C 180,E1 24815.517,E2 24815.517} C_VEL
LIN {X 0,Y 549.892,Z 431.198,A -85,B 0,C 180,E1 24814.53,E2 24814.53} C_VEL
LIN {X 0,Y 555.54,Z 438.401,A -85,B 0,C 180,E1 24813.143,E2 24813.143} C_VEL
LIN {X 0,Y 560.036,Z 444.072,A -85,B 0,C 180,E1 24812.105,E2 24812.105} C_VEL
LIN {X 0,Y 567.879,Z 454.217,A -85,B 0,C 180,E1 24810.403,E2 24810.403} C_VEL
LIN {X 0,Y 579.355,Z 469.745,A -85,B 0,C 180,E1 24808.122,E2 24808.122} C_VEL
LIN {X 0,Y 592.251,Z 488.308,A -85,B 0,C 180,E1 24805.792,E2 24805.792} C_VEL
LIN {X 0,Y 604.509,Z 507.225,A -85,B 0,C 180,E1 24803.759,E2 24803.759} C_VEL
LIN {X 0,Y 596.63,Z 727.133,A -85,B 0,C 180,E1 24800.54,E2 24800.54} C_VEL
LIN {X 0,Y 590.599,Z 901.818,A -85,B 0,C 180,E1 24798.012,E2 24798.012} C_VEL
LIN {X 0,Y 588.938,Z 926.507,A -85,B 0,C 180,E1 24797.56,E2 24797.56} C_VEL
LIN {X 0,Y 586.298,Z 954.866,A -85,B 0,C 180,E1 24796.851,E2 24796.851} C_VEL
LIN {X 0,Y 583.781,Z 977.073,A -85,B 0,C 180,E1 24796.147,E2 24796.147} C_VEL
LIN {X 0,Y 581.109,Z 997.894,A -85,B 0,C 180,E1 24795.359,E2 24795.359} C_VEL
LIN {X 0,Y 578.224,Z 1018.315,A -85,B 0,C 180,E1 24794.458,E2 24794.458} C_VEL
LIN {X 0,Y 574.361,Z 1043.396,A -85,B 0,C 180,E1 24793.173,E2 24793.173} C_VEL
LIN {X 0,Y 570.378,Z 1066.468,A -85,B 0,C 180,E1 24791.774,E2 24791.774} C_VEL
LIN {X 0,Y 566.951,Z 1085.422,A -85,B 0,C 180,E1 24790.47,E2 24790.47} C_VEL
LIN {X 0,Y 563.622,Z 1103.203,A -85,B 0,C 180,E1 24789.103,E2 24789.103} C_VEL
LIN {X 0,Y 560.24,Z 1120.9,A -85,B 0,C 180,E1 24787.586,E2 24787.586} C_VEL
LIN {X 0,Y 556.462,Z 1140.681,A -85,B 0,C 180,E1 24785.69,E2 24785.69} C_VEL
LIN {X 0,Y 552.546,Z 1160.552,A -85,B 0,C 180,E1 24783.503,E2 24783.503} C_VEL
LIN {X 0,Y 549.555,Z 1175.791,A -85,B 0,C 180,E1 24781.605,E2 24781.605} C_VEL
LIN {X 0,Y 546.966,Z 1189.572,A -85,B 0,C 180,E1 24779.7,E2 24779.7} C_VEL
LIN {X 0,Y 544.606,Z 1202.744,A -85,B 0,C 180,E1 24777.682,E2 24777.682} C_VEL
LIN {X 0,Y 542.095,Z 1217.861,A -85,B 0,C 180,E1 24775.089,E2 24775.089} C_VEL
LIN {X 0,Y 540.066,Z 1231.208,A -85,B 0,C 180,E1 24772.424,E2 24772.424} C_VEL
LIN {X 0,Y 538.732,Z 1241.477,A -85,B 0,C 180,E1 24770.092,E2 24770.092} C_VEL
LIN {X 0,Y 537.698,Z 1250.495,A -85,B 0,C 180,E1 24767.76,E2 24767.76} C_VEL
LIN {X 0,Y 536.848,Z 1259.993,A -85,B 0,C 180,E1 24764.898,E2 24764.898} C_VEL
LIN {X 0,Y 536.335,Z 1267.281,A -85,B 0,C 180,E1 24762.166,E2 24762.166} C_VEL
LIN {X 0,Y 536.062,Z 1272.486,A -85,B 0,C 180,E1 24759.777,E2 24759.777} C_VEL
LIN {X 0,Y 535.96,Z 1276.359,A -85,B 0,C 180,E1 24757.508,E2 24757.508} C_VEL
LIN {X 0,Y 535.923,Z 1279.317,A -85,B 0,C 180,E1 24755.143,E2 24755.143} C_VEL
LIN {X 0,Y 535.907,Z 1281.283,A -85,B 0,C 180,E1 24752.571,E2 24752.571} C_VEL
LIN {X 0,Y 535.878,Z 1281.94,A -85,B 0,C 180,E1 24749.684,E2 24749.684} C_VEL
LIN {X 0,Y 535.91,Z 1281.085,A -85,B 0,C 180,E1 24747.118,E2 24747.118} C_VEL
LIN {X 0,Y 535.925,Z 1279.213,A -85,B 0,C 180,E1 24744.76,E2 24744.76} C_VEL
LIN {X 0,Y 535.96,Z 1276.373,A -85,B 0,C 180,E1 24742.502,E2 24742.502} C_VEL
LIN {X 0,Y 536.061,Z 1272.505,A -85,B 0,C 180,E1 24740.233,E2 24740.233} C_VEL
LIN {X 0,Y 536.322,Z 1267.558,A -85,B 0,C 180,E1 24737.953,E2 24737.953} C_VEL
LIN {X 0,Y 536.775,Z 1260.631,A -85,B 0,C 180,E1 24735.331,E2 24735.331} C_VEL
LIN {X 0,Y 537.651,Z 1250.936,A -85,B 0,C 180,E1 24732.36,E2 24732.36} C_VEL
LIN {X 0,Y 538.734,Z 1241.479,A -85,B 0,C 180,E1 24729.908,E2 24729.908} C_VEL
LIN {X 0,Y 540.059,Z 1231.261,A -85,B 0,C 180,E1 24727.586,E2 24727.586} C_VEL
LIN {X 0,Y 542.1,Z 1217.833,A -85,B 0,C 180,E1 24724.905,E2 24724.905} C_VEL
LIN {X 0,Y 544.596,Z 1202.809,A -85,B 0,C 180,E1 24722.328,E2 24722.328} C_VEL
LIN {X 0,Y 547.017,Z 1189.274,A -85,B 0,C 180,E1 24720.256,E2 24720.256} C_VEL
LIN {X 0,Y 549.888,Z 1174.177,A -85,B 0,C 180,E1 24718.183,E2 24718.183} C_VEL
LIN {X 0,Y 553.965,Z 1153.392,A -85,B 0,C 180,E1 24715.671,E2 24715.671} C_VEL
LIN {X 0,Y 557.234,Z 1136.446,A -85,B 0,C 180,E1 24713.89,E2 24713.89} C_VEL
LIN {X 0,Y 560.505,Z 1119.448,A -85,B 0,C 180,E1 24712.283,E2 24712.283} C_VEL
LIN {X 0,Y 563.976,Z 1101.291,A -85,B 0,C 180,E1 24710.742,E2 24710.742} C_VEL
LIN {X 0,Y 568.276,Z 1078.322,A -85,B 0,C 180,E1 24709.011,E2 24709.011} C_VEL
LIN {X 0,Y 572.422,Z 1054.483,A -85,B 0,C 180,E1 24707.477,E2 24707.477} C_VEL
LIN {X 0,Y 575.705,Z 1034.478,A -85,B 0,C 180,E1 24706.349,E2 24706.349} C_VEL
LIN {X 0,Y 578.844,Z 1013.974,A -85,B 0,C 180,E1 24705.338,E2 24705.338} C_VEL
LIN {X 0,Y 582.338,Z 989.084,A -85,B 0,C 180,E1 24704.285,E2 24704.285} C_VEL
LIN {X 0,Y 585.48,Z 962.357,A -85,B 0,C 180,E1 24703.371,E2 24703.371} C_VEL
LIN {X 0,Y 587.691,Z 940.539,A -85,B 0,C 180,E1 24702.768,E2 24702.768} C_VEL
LIN {X 0,Y 589.476,Z 919.158,A -85,B 0,C 180,E1 24702.294,E2 24702.294} C_VEL
LIN {X 0,Y 590.886,Z 895.976,A -85,B 0,C 180,E1 24701.896,E2 24701.896} C_VEL
LIN {X 0,Y 598.448,Z 674.473,A -85,B 0,C 180,E1 24698.696,E2 24698.696} C_VEL
LIN {X 0,Y 604.405,Z 507.1,A -85,B 0,C 180,E1 24696.229,E2 24696.229} C_VEL
LIN {X 0,Y 592.219,Z 488.295,A -85,B 0,C 180,E1 24694.21,E2 24694.21} C_VEL
LIN {X 0,Y 579.075,Z 469.402,A -85,B 0,C 180,E1 24691.837,E2 24691.837} C_VEL
LIN {X 0,Y 568.575,Z 455.249,A -85,B 0,C 180,E1 24689.76,E2 24689.76} C_VEL
LIN {X 0,Y 562.13,Z 446.862,A -85,B 0,C 180,E1 24688.384,E2 24688.384} C_VEL
LIN {X 0,Y 557.987,Z 441.536,A -85,B 0,C 180,E1 24687.451,E2 24687.451} C_VEL
LIN {X 0,Y 553.278,Z 435.585,A -85,B 0,C 180,E1 24686.338,E2 24686.338} C_VEL
LIN {X 0,Y 549.022,Z 430.372,A -85,B 0,C 180,E1 24685.282,E2 24685.282} C_VEL
LIN {X 0,Y 544.754,Z 425.108,A -85,B 0,C 180,E1 24684.162,E2 24684.162} C_VEL
LIN {X 0,Y 541.353,Z 421.067,A -85,B 0,C 180,E1 24683.225,E2 24683.225} C_VEL
LIN {X 0,Y 540.269,Z 419.344,A -85,B 0,C 180,E1 24682.871,E2 24682.871} C_VEL
LIN {X 0,Y 538.112,Z 416.223,A -85,B 0,C 180,E1 24681.816,E2 24681.816} C_VEL
LIN {X 0,Y 537.577,Z 414.221,A -85,B 0,C 180,E1 24681.266,E2 24681.266} C_VEL
LIN {X 0,Y 537.554,Z 414.258,A -85,B 0,C 180,E1 24678.097,E2 24678.097} C_VEL
LIN {X 0,Y 537.531,Z 414.213,A -85,B 0,C 180,E1 24674.654,E2 24674.654} C_VEL
LIN {X 0,Y 537.588,Z 414.259,A -85,B 0,C 180,E1 24671.463,E2 24671.463} C_VEL
LIN {X 0,Y 537.516,Z 414.221,A -85,B 0,C 180,E1 24668.235,E2 24668.235} C_VEL
LIN {X 0,Y 537.579,Z 414.241,A -85,B 0,C 180,E1 24665.015,E2 24665.015} C_VEL
LIN {X 0,Y 537.532,Z 414.227,A -85,B 0,C 180,E1 24661.812,E2 24661.812} C_VEL
LIN {X 0,Y 537.545,Z 414.228,A -85,B 0,C 180,E1 24658.401,E2 24658.401} C_VEL
LIN {X 0,Y 537.582,Z 414.236,A -85,B 0,C 180,E1 24655.199,E2 24655.199} C_VEL
LIN {X 0,Y 537.543,Z 414.22,A -85,B 0,C 180,E1 24651.981,E2 24651.981} C_VEL
LIN {X 0,Y 537.615,Z 414.249,A -85,B 0,C 180,E1 24648.739,E2 24648.739} C_VEL
LIN {X 0,Y 537.551,Z 414.212,A -85,B 0,C 180,E1 24645.567,E2 24645.567} C_VEL
LIN {X 0,Y 537.596,Z 414.267,A -85,B 0,C 180,E1 24642.202,E2 24642.202} C_VEL
LIN {X 0,Y 537.588,Z 414.21,A -85,B 0,C 180,E1 24638.963,E2 24638.963} C_VEL
LIN {X 0,Y 537.582,Z 414.363,A -85,B 0,C 180,E1 24637.442,E2 24637.442} C_VEL
LIN {X 0,Y 538.51,Z 417.136,A -85,B 0,C 180,E1 24637.108,E2 24637.108} C_VEL
LIN {X 0,Y 540.944,Z 419.792,A -85,B 0,C 180,E1 24636.41,E2 24636.41} C_VEL
LIN {X 0,Y 543.19,Z 421.201,A -85,B 0,C 180,E1 24635.822,E2 24635.822} C_VEL
LIN {X 0,Y 545.164,Z 424.636,A -85,B 0,C 180,E1 24635.251,E2 24635.251} C_VEL
LIN {X 0,Y 548.725,Z 427.691,A -85,B 0,C 180,E1 24634.356,E2 24634.356} C_VEL
LIN {X 0,Y 551.34,Z 431.528,A -85,B 0,C 180,E1 24633.678,E2 24633.678} C_VEL
LIN {X 0,Y 554.073,Z 433.957,A -85,B 0,C 180,E1 24633.037,E2 24633.037} C_VEL
LIN {X 0,Y 557.252,Z 438.208,A -85,B 0,C 180,E1 24632.278,E2 24632.278} C_VEL
LIN {X 0,Y 559.457,Z 440.383,A -85,B 0,C 180,E1 24631.788,E2 24631.788} C_VEL
LIN {X 0,Y 563.026,Z 444.72,A -85,B 0,C 180,E1 24630.999,E2 24630.999} C_VEL
LIN {X 0,Y 569.542,Z 452.732,A -85,B 0,C 180,E1 24629.628,E2 24629.628} C_VEL
LIN {X 0,Y 577.845,Z 462.984,A -85,B 0,C 180,E1 24627.999,E2 24627.999} C_VEL
LIN {X 0,Y 589.921,Z 478.706,A -85,B 0,C 180,E1 24625.814,E2 24625.814} C_VEL
LIN {X 0,Y 602.898,Z 496.599,A -85,B 0,C 180,E1 24623.666,E2 24623.666} C_VEL
LIN {X 0,Y 604.309,Z 498.89,A -85,B 0,C 180,E1 24623.438,E2 24623.438} C_VEL
LIN {X 0,Y 596.454,Z 715.667,A -85,B 0,C 180,E1 24620.264,E2 24620.264} C_VEL
LIN {X 0,Y 590.823,Z 876.03,A -85,B 0,C 180,E1 24617.939,E2 24617.939} C_VEL
LIN {X 0,Y 590.281,Z 885.968,A -85,B 0,C 180,E1 24617.774,E2 24617.774} C_VEL
LIN {X 0,Y 588.981,Z 893.587,A -85,B 0,C 180,E1 24617.707,E2 24617.707} C_VEL
LIN {X 0,Y 583.879,Z 910.737,A -85,B 0,C 180,E1 24617.733,E2 24617.733} C_VEL
LIN {X 0,Y 582.151,Z 919.351,A -85,B 0,C 180,E1 24617.612,E2 24617.612} C_VEL
LIN {X 0,Y 582.042,Z 920.423,A -85,B 0,C 180,E1 24617.586,E2 24617.586} C_VEL
LIN {X 0,Y 578.927,Z 948.134,A -85,B 0,C 180,E1 24616.733,E2 24616.733} C_VEL
LIN {X 0,Y 576.101,Z 969.489,A -85,B 0,C 180,E1 24615.924,E2 24615.924} C_VEL
LIN {X 0,Y 573.18,Z 989.272,A -85,B 0,C 180,E1 24615.048,E2 24615.048} C_VEL
LIN {X 0,Y 569.832,Z 1009.728,A -85,B 0,C 180,E1 24614.007,E2 24614.007} C_VEL
LIN {X 0,Y 565.644,Z 1033.579,A -85,B 0,C 180,E1 24612.603,E2 24612.603} C_VEL
LIN {X 0,Y 561.214,Z 1056.278,A -85,B 0,C 180,E1 24611.027,E2 24611.027} C_VEL
LIN {X 0,Y 557.523,Z 1074.419,A -85,B 0,C 180,E1 24609.602,E2 24609.602} C_VEL
LIN {X 0,Y 553.929,Z 1091.594,A -85,B 0,C 180,E1 24608.092,E2 24608.092} C_VEL
LIN {X 0,Y 550.144,Z 1109.52,A -85,B 0,C 180,E1 24606.327,E2 24606.327} C_VEL
LIN {X 0,Y 545.653,Z 1130.473,A -85,B 0,C 180,E1 24603.972,E2 24603.972} C_VEL
LIN {X 0,Y 541.946,Z 1148.095,A -85,B 0,C 180,E1 24601.716,E2 24601.716} C_VEL
LIN {X 0,Y 538.877,Z 1163.978,A -85,B 0,C 180,E1 24599.445,E2 24599.445} C_VEL
LIN {X 0,Y 535.759,Z 1180.611,A -85,B 0,C 180,E1 24596.722,E2 24596.722} C_VEL
LIN {X 0,Y 533.659,Z 1193.008,A -85,B 0,C 180,E1 24594.412,E2 24594.412} C_VEL
LIN {X 0,Y 532.003,Z 1203.633,A -85,B 0,C 180,E1 24592.189,E2 24592.189} C_VEL
LIN {X 0,Y 530.483,Z 1215.035,A -85,B 0,C 180,E1 24589.482,E2 24589.482} C_VEL
LIN {X 0,Y 529.345,Z 1225.321,A -85,B 0,C 180,E1 24586.566,E2 24586.566} C_VEL
LIN {X 0,Y 528.686,Z 1232.333,A -85,B 0,C 180,E1 24584.227,E2 24584.227} C_VEL
LIN {X 0,Y 528.331,Z 1237.963,A -85,B 0,C 180,E1 24582.01,E2 24582.01} C_VEL
LIN {X 0,Y 528.061,Z 1242.831,A -85,B 0,C 180,E1 24579.696,E2 24579.696} C_VEL
LIN {X 0,Y 527.963,Z 1246.624,A -85,B 0,C 180,E1 24577.394,E2 24577.394} C_VEL
LIN {X 0,Y 527.922,Z 1249.618,A -85,B 0,C 180,E1 24574.884,E2 24574.884} C_VEL
LIN {X 0,Y 527.91,Z 1251.591,A -85,B 0,C 180,E1 24571.949,E2 24571.949} C_VEL
LIN {X 0,Y 527.866,Z 1251.88,A -85,B 0,C 180,E1 24569.344,E2 24569.344} C_VEL
LIN {X 0,Y 527.909,Z 1251.04,A -85,B 0,C 180,E1 24566.955,E2 24566.955} C_VEL
LIN {X 0,Y 527.926,Z 1249.134,A -85,B 0,C 180,E1 24564.561,E2 24564.561} C_VEL
LIN {X 0,Y 527.969,Z 1246.103,A -85,B 0,C 180,E1 24562.158,E2 24562.158} C_VEL
LIN {X 0,Y 528.162,Z 1241.534,A -85,B 0,C 180,E1 24559.524,E2 24559.524} C_VEL
LIN {X 0,Y 528.569,Z 1234.369,A -85,B 0,C 180,E1 24556.429,E2 24556.429} C_VEL
LIN {X 0,Y 529.135,Z 1227.339,A -85,B 0,C 180,E1 24553.981,E2 24553.981} C_VEL
LIN {X 0,Y 529.964,Z 1219.426,A -85,B 0,C 180,E1 24551.627,E2 24551.627} C_VEL
LIN {X 0,Y 531.103,Z 1210.303,A -85,B 0,C 180,E1 24549.267,E2 24549.267} C_VEL
LIN {X 0,Y 532.935,Z 1197.767,A -85,B 0,C 180,E1 24546.441,E2 24546.441} C_VEL
LIN {X 0,Y 535.236,Z 1183.629,A -85,B 0,C 180,E1 24543.728,E2 24543.728} C_VEL
LIN {X 0,Y 537.392,Z 1171.49,A -85,B 0,C 180,E1 24541.653,E2 24541.653} C_VEL
LIN {X 0,Y 540.094,Z 1157.54,A -85,B 0,C 180,E1 24539.515,E2 24539.515} C_VEL
LIN {X 0,Y 543.922,Z 1138.712,A -85,B 0,C 180,E1 24536.958,E2 24536.958} C_VEL
LIN {X 0,Y 547.56,Z 1121.422,A -85,B 0,C 180,E1 24534.882,E2 24534.882} C_VEL
LIN {X 0,Y 550.985,Z 1105.387,A -85,B 0,C 180,E1 24533.159,E2 24533.159} C_VEL
LIN {X 0,Y 554.575,Z 1088.511,A -85,B 0,C 180,E1 24531.532,E2 24531.532} C_VEL
LIN {X 0,Y 559.2,Z 1066.574,A -85,B 0,C 180,E1 24529.66,E2 24529.66} C_VEL
LIN {X 0,Y 563.439,Z 1044.952,A -85,B 0,C 180,E1 24528.073,E2 24528.073} C_VEL
LIN {X 0,Y 567.031,Z 1025.673,A -85,B 0,C 180,E1 24526.825,E2 24526.825} C_VEL
LIN {X 0,Y 570.483,Z 1005.841,A -85,B 0,C 180,E1 24525.694,E2 24525.694} C_VEL
LIN {X 0,Y 574.314,Z 982.088,A -85,B 0,C 180,E1 24524.522,E2 24524.522} C_VEL
LIN {X 0,Y 577.931,Z 956.107,A -85,B 0,C 180,E1 24523.463,E2 24523.463} C_VEL
LIN {X 0,Y 580.54,Z 934.246,A -85,B 0,C 180,E1 24522.724,E2 24522.724} C_VEL
LIN {X 0,Y 582.703,Z 913.245,A -85,B 0,C 180,E1 24522.142,E2 24522.142} C_VEL
LIN {X 0,Y 584.502,Z 891.585,A -85,B 0,C 180,E1 24521.659,E2 24521.659} C_VEL
LIN {X 0,Y 586.117,Z 864.147,A -85,B 0,C 180,E1 24521.196,E2 24521.196} C_VEL
LIN {X 0,Y 594.121,Z 641.692,A -85,B 0,C 180,E1 24517.961,E2 24517.961} C_VEL
LIN {X 0,Y 599.383,Z 502.795,A -85,B 0,C 180,E1 24515.9,E2 24515.9} C_VEL
LIN {X 0,Y 585.95,Z 484.115,A -85,B 0,C 180,E1 24513.624,E2 24513.624} C_VEL
LIN {X 0,Y 573.946,Z 468.435,A -85,B 0,C 180,E1 24511.393,E2 24511.393} C_VEL
LIN {X 0,Y 564.595,Z 456.866,A -85,B 0,C 180,E1 24509.494,E2 24509.494} C_VEL
LIN {X 0,Y 560.441,Z 451.755,A -85,B 0,C 180,E1 24508.593,E2 24508.593} C_VEL
LIN {X 0,Y 555.788,Z 446.184,A -85,B 0,C 180,E1 24507.539,E2 24507.539} C_VEL
LIN {X 0,Y 552.184,Z 441.902,A -85,B 0,C 180,E1 24506.685,E2 24506.685} C_VEL
LIN {X 0,Y 551.012,Z 440.451,A -85,B 0,C 180,E1 24506.397,E2 24506.397} C_VEL
LIN {X 0,Y 547.516,Z 436.694,A -85,B 0,C 180,E1 24505.531,E2 24505.531} C_VEL
LIN {X 0,Y 546.058,Z 434.529,A -85,B 0,C 180,E1 24505.139,E2 24505.139} C_VEL
LIN {X 0,Y 542.764,Z 431.524,A -85,B 0,C 180,E1 24504.285,E2 24504.285} C_VEL
LIN {X 0,Y 540.802,Z 428.344,A -85,B 0,C 180,E1 24503.712,E2 24503.712} C_VEL
LIN {X 0,Y 537.55,Z 425.923,A -85,B 0,C 180,E1 24502.82,E2 24502.82} C_VEL
LIN {X 0,Y 535.567,Z 422.502,A -85,B 0,C 180,E1 24502.185,E2 24502.185} C_VEL
LIN {X 0,Y 535.175,Z 421.852,A -85,B 0,C 180,E1 24502.058,E2 24502.058} C_VEL
LIN {X 0,Y 531.94,Z 419.863,A -85,B 0,C 180,E1 24501.098,E2 24501.098} C_VEL
LIN {X 0,Y 530.151,Z 417.08,A -85,B 0,C 180,E1 24500.479,E2 24500.479} C_VEL
LIN {X 0,Y 529.672,Z 415.191,A -85,B 0,C 180,E1 24500.241,E2 24500.241} C_VEL
LIN {X 0,Y 529.668,Z 415.232,A -85,B 0,C 180,E1 24496.838,E2 24496.838} C_VEL
LIN {X 0,Y 529.675,Z 415.208,A -85,B 0,C 180,E1 24493.315,E2 24493.315} C_VEL
LIN {X 0,Y 529.673,Z 415.196,A -85,B 0,C 180,E1 24489.892,E2 24489.892} C_VEL
LIN {X 0,Y 529.665,Z 415.241,A -85,B 0,C 180,E1 24486.504,E2 24486.504} C_VEL
LIN {X 0,Y 529.67,Z 415.184,A -85,B 0,C 180,E1 24483.03,E2 24483.03} C_VEL
LIN {X 0,Y 529.683,Z 415.252,A -85,B 0,C 180,E1 24479.567,E2 24479.567} C_VEL
LIN {X 0,Y 529.655,Z 415.188,A -85,B 0,C 180,E1 24476.103,E2 24476.103} C_VEL
LIN {X 0,Y 529.675,Z 415.222,A -85,B 0,C 180,E1 24472.625,E2 24472.625} C_VEL
LIN {X 0,Y 529.68,Z 415.211,A -85,B 0,C 180,E1 24469.119,E2 24469.119} C_VEL
LIN {X 0,Y 529.652,Z 415.198,A -85,B 0,C 180,E1 24465.793,E2 24465.793} C_VEL
LIN {X 0,Y 529.677,Z 415.254,A -85,B 0,C 180,E1 24462.306,E2 24462.306} C_VEL
LIN {X 0,Y 529.695,Z 415.314,A -85,B 0,C 180,E1 24460.653,E2 24460.653} C_VEL
LIN {X 0,Y 531.193,Z 419.014,A -85,B 0,C 180,E1 24459.563,E2 24459.563} C_VEL
LIN {X 0,Y 533.768,Z 421.616,A -85,B 0,C 180,E1 24458.747,E2 24458.747} C_VEL
LIN {X 0,Y 536.686,Z 425.483,A -85,B 0,C 180,E1 24457.835,E2 24457.835} C_VEL
LIN {X 0,Y 538.772,Z 427.481,A -85,B 0,C 180,E1 24457.235,E2 24457.235} C_VEL
LIN {X 0,Y 542.058,Z 431.86,A -85,B 0,C 180,E1 24456.289,E2 24456.289} C_VEL
LIN {X 0,Y 544.248,Z 434.281,A -85,B 0,C 180,E1 24455.699,E2 24455.699} C_VEL
LIN {X 0,Y 552.879,Z 445.129,A -85,B 0,C 180,E1 24453.496,E2 24453.496} C_VEL
LIN {X 0,Y 558.002,Z 451.797,A -85,B 0,C 180,E1 24452.29,E2 24452.29} C_VEL
LIN {X 0,Y 564.951,Z 460.786,A -85,B 0,C 180,E1 24450.759,E2 24450.759} C_VEL
LIN {X 0,Y 576.63,Z 476.829,A -85,B 0,C 180,E1 24448.392,E2 24448.392} C_VEL
LIN {X 0,Y 589.661,Z 495.76,A -85,B 0,C 180,E1 24446.002,E2 24446.002} C_VEL
LIN {X 0,Y 599.61,Z 511.46,A -85,B 0,C 180,E1 24444.313,E2 24444.313} C_VEL
LIN {X 0,Y 591.253,Z 734.845,A -85,B 0,C 180,E1 24441.027,E2 24441.027} C_VEL
LIN {X 0,Y 585.238,Z 901.67,A -85,B 0,C 180,E1 24438.597,E2 24438.597} C_VEL
LIN {X 0,Y 583.475,Z 926.903,A -85,B 0,C 180,E1 24438.132,E2 24438.132} C_VEL
LIN {X 0,Y 580.759,Z 954.779,A -85,B 0,C 180,E1 24437.43,E2 24437.43} C_VEL
LIN {X 0,Y 578.168,Z 976.809,A -85,B 0,C 180,E1 24436.729,E2 24436.729} C_VEL
LIN {X 0,Y 575.411,Z 997.498,A -85,B 0,C 180,E1 24435.944,E2 24435.944} C_VEL
LIN {X 0,Y 572.544,Z 1016.907,A -85,B 0,C 180,E1 24435.089,E2 24435.089} C_VEL
LIN {X 0,Y 568.971,Z 1039.08,A -85,B 0,C 180,E1 24433.963,E2 24433.963} C_VEL
LIN {X 0,Y 564.335,Z 1065.457,A -85,B 0,C 180,E1 24432.386,E2 24432.386} C_VEL
LIN {X 0,Y 560.606,Z 1085.196,A -85,B 0,C 180,E1 24431.022,E2 24431.022} C_VEL
LIN {X 0,Y 557.003,Z 1103.603,A -85,B 0,C 180,E1 24429.592,E2 24429.592} C_VEL
LIN {X 0,Y 553.377,Z 1121.713,A -85,B 0,C 180,E1 24428.019,E2 24428.019} C_VEL
LIN {X 0,Y 549.053,Z 1143.277,A -85,B 0,C 180,E1 24425.905,E2 24425.905} C_VEL
LIN {X 0,Y 545.15,Z 1162.288,A -85,B 0,C 180,E1 24423.766,E2 24423.766} C_VEL
LIN {X 0,Y 542.429,Z 1175.789,A -85,B 0,C 180,E1 24422.069,E2 24422.069} C_VEL
LIN {X 0,Y 539.588,Z 1190.037,A -85,B 0,C 180,E1 24420.073,E2 24420.073} C_VEL
LIN {X 0,Y 537.049,Z 1203.443,A -85,B 0,C 180,E1 24417.985,E2 24417.985} C_VEL
LIN {X 0,Y 534.33,Z 1218.948,A -85,B 0,C 180,E1 24415.259,E2 24415.259} C_VEL
LIN {X 0,Y 532.286,Z 1231.721,A -85,B 0,C 180,E1 24412.653,E2 24412.653} C_VEL
LIN {X 0,Y 530.879,Z 1241.959,A -85,B 0,C 180,E1 24410.281,E2 24410.281} C_VEL
LIN {X 0,Y 529.704,Z 1251.709,A -85,B 0,C 180,E1 24407.697,E2 24407.697} C_VEL
LIN {X 0,Y 528.793,Z 1261.216,A -85,B 0,C 180,E1 24404.682,E2 24404.682} C_VEL
LIN {X 0,Y 528.353,Z 1267.534,A -85,B 0,C 180,E1 24402.241,E2 24402.241} C_VEL
LIN {X 0,Y 528.085,Z 1272.483,A -85,B 0,C 180,E1 24399.926,E2 24399.926} C_VEL
LIN {X 0,Y 527.961,Z 1276.357,A -85,B 0,C 180,E1 24397.623,E2 24397.623} C_VEL
LIN {X 0,Y 527.924,Z 1279.201,A -85,B 0,C 180,E1 24395.33,E2 24395.33} C_VEL
LIN {X 0,Y 527.909,Z 1281.079,A -85,B 0,C 180,E1 24392.936,E2 24392.936} C_VEL
LIN {X 0,Y 527.877,Z 1281.938,A -85,B 0,C 180,E1 24390.331,E2 24390.331} C_VEL
LIN {X 0,Y 527.909,Z 1281.289,A -85,B 0,C 180,E1 24387.4,E2 24387.4} C_VEL
LIN {X 0,Y 527.925,Z 1279.324,A -85,B 0,C 180,E1 24384.789,E2 24384.789} C_VEL
LIN {X 0,Y 527.962,Z 1276.53,A -85,B 0,C 180,E1 24382.497,E2 24382.497} C_VEL
LIN {X 0,Y 528.069,Z 1272.708,A -85,B 0,C 180,E1 24380.194,E2 24380.194} C_VEL
LIN {X 0,Y 528.339,Z 1267.812,A -85,B 0,C 180,E1 24377.879,E2 24377.879} C_VEL
LIN {X 0,Y 528.733,Z 1261.775,A -85,B 0,C 180,E1 24375.524,E2 24375.524} C_VEL
LIN {X 0,Y 529.542,Z 1253.33,A -85,B 0,C 180,E1 24372.762,E2 24372.762} C_VEL
LIN {X 0,Y 530.814,Z 1242.463,A -85,B 0,C 180,E1 24369.842,E2 24369.842} C_VEL
LIN {X 0,Y 532.2,Z 1232.288,A -85,B 0,C 180,E1 24367.47,E2 24367.47} C_VEL
LIN {X 0,Y 534.016,Z 1220.727,A -85,B 0,C 180,E1 24365.091,E2 24365.091} C_VEL
LIN {X 0,Y 536.923,Z 1204.208,A -85,B 0,C 180,E1 24362.14,E2 24362.14} C_VEL
LIN {X 0,Y 539.513,Z 1190.41,A -85,B 0,C 180,E1 24359.981,E2 24359.981} C_VEL
LIN {X 0,Y 542.3,Z 1176.388,A -85,B 0,C 180,E1 24358.011,E2 24358.011} C_VEL
LIN {X 0,Y 544.938,Z 1163.314,A -85,B 0,C 180,E1 24356.357,E2 24356.357} C_VEL
LIN {X 0,Y 548.251,Z 1146.97,A -85,B 0,C 180,E1 24354.496,E2 24354.496} C_VEL
LIN {X 0,Y 552.694,Z 1125.334,A -85,B 0,C 180,E1 24352.312,E2 24352.312} C_VEL
LIN {X 0,Y 556.719,Z 1105.07,A -85,B 0,C 180,E1 24350.53,E2 24350.53} C_VEL
LIN {X 0,Y 560.307,Z 1086.759,A -85,B 0,C 180,E1 24349.095,E2 24349.095} C_VEL
LIN {X 0,Y 563.865,Z 1067.979,A -85,B 0,C 180,E1 24347.782,E2 24347.782} C_VEL
LIN {X 0,Y 567.448,Z 1048.12,A -85,B 0,C 180,E1 24346.551,E2 24346.551} C_VEL
LIN {X 0,Y 571.69,Z 1022.816,A -85,B 0,C 180,E1 24345.192,E2 24345.192} C_VEL
LIN {X 0,Y 574.995,Z 1000.448,A -85,B 0,C 180,E1 24344.176,E2 24344.176} C_VEL
LIN {X 0,Y 577.85,Z 979.307,A -85,B 0,C 180,E1 24343.359,E2 24343.359} C_VEL
LIN {X 0,Y 580.351,Z 958.381,A -85,B 0,C 180,E1 24342.678,E2 24342.678} C_VEL
LIN {X 0,Y 582.556,Z 936.812,A -85,B 0,C 180,E1 24342.098,E2 24342.098} C_VEL
LIN {X 0,Y 584.747,Z 910.628,A -85,B 0,C 180,E1 24341.549,E2 24341.549} C_VEL
LIN {X 0,Y 586.496,Z 870.289,A -85,B 0,C 180,E1 24340.935,E2 24340.935} C_VEL
LIN {X 0,Y 594.338,Z 649.882,A -85,B 0,C 180,E1 24337.733,E2 24337.733} C_VEL
LIN {X 0,Y 599.457,Z 511.137,A -85,B 0,C 180,E1 24335.665,E2 24335.665} C_VEL
LIN {X 0,Y 587.307,Z 492.431,A -85,B 0,C 180,E1 24333.595,E2 24333.595} C_VEL
LIN {X 0,Y 575.44,Z 475.136,A -85,B 0,C 180,E1 24331.389,E2 24331.389} C_VEL
LIN {X 0,Y 564.239,Z 459.91,A -85,B 0,C 180,E1 24329.107,E2 24329.107} C_VEL
LIN {X 0,Y 558.746,Z 452.868,A -85,B 0,C 180,E1 24327.902,E2 24327.902} C_VEL
LIN {X 0,Y 555.384,Z 448.449,A -85,B 0,C 180,E1 24327.126,E2 24327.126} C_VEL
LIN {X 0,Y 550.637,Z 442.403,A -85,B 0,C 180,E1 24325.982,E2 24325.982} C_VEL
LIN {X 0,Y 546.535,Z 437.328,A -85,B 0,C 180,E1 24324.942,E2 24324.942} C_VEL
LIN {X 0,Y 542.692,Z 432.49,A -85,B 0,C 180,E1 24323.913,E2 24323.913} C_VEL
LIN {X 0,Y 539.077,Z 428.08,A -85,B 0,C 180,E1 24322.895,E2 24322.895} C_VEL
LIN {X 0,Y 537.972,Z 426.63,A -85,B 0,C 180,E1 24322.57,E2 24322.57} C_VEL
LIN {X 0,Y 534.587,Z 423.005,A -85,B 0,C 180,E1 24321.564,E2 24321.564} C_VEL
LIN {X 0,Y 533.172,Z 420.907,A -85,B 0,C 180,E1 24321.105,E2 24321.105} C_VEL
LIN {X 0,Y 530.564,Z 418.109,A -85,B 0,C 180,E1 24320.174,E2 24320.174} C_VEL
LIN {X 0,Y 529.643,Z 415.204,A -85,B 0,C 180,E1 24319.292,E2 24319.292} C_VEL
LIN {X 0,Y 529.598,Z 415.219,A -85,B 0,C 180,E1 24316.226,E2 24316.226} C_VEL
LIN {X 0,Y 529.602,Z 415.241,A -85,B 0,C 180,E1 24312.762,E2 24312.762} C_VEL
LIN {X 0,Y 529.625,Z 415.196,A -85,B 0,C 180,E1 24309.563,E2 24309.563} C_VEL
LIN {X 0,Y 529.584,Z 415.265,A -85,B 0,C 180,E1 24306.287,E2 24306.287} C_VEL
LIN {X 0,Y 529.642,Z 415.19,A -85,B 0,C 180,E1 24303.03,E2 24303.03} C_VEL
LIN {X 0,Y 529.602,Z 415.262,A -85,B 0,C 180,E1 24299.784,E2 24299.784} C_VEL
LIN {X 0,Y 529.605,Z 415.199,A -85,B 0,C 180,E1 24296.32,E2 24296.32} C_VEL
LIN {X 0,Y 529.66,Z 415.234,A -85,B 0,C 180,E1 24293.061,E2 24293.061} C_VEL
LIN {X 0,Y 529.607,Z 415.208,A -85,B 0,C 180,E1 24289.777,E2 24289.777} C_VEL
LIN {X 0,Y 529.66,Z 415.21,A -85,B 0,C 180,E1 24286.462,E2 24286.462} C_VEL
LIN {X 0,Y 529.627,Z 415.225,A -85,B 0,C 180,E1 24283.324,E2 24283.324} C_VEL
LIN {X 0,Y 529.634,Z 415.197,A -85,B 0,C 180,E1 24279.904,E2 24279.904} C_VEL
LIN {X 0,Y 529.641,Z 415.342,A -85,B 0,C 180,E1 24279.601,E2 24279.601} C_VEL
LIN {X 0,Y 530.51,Z 417.979,A -85,B 0,C 180,E1 24279.247,E2 24279.247} C_VEL
LIN {X 0,Y 532.877,Z 420.651,A -85,B 0,C 180,E1 24278.479,E2 24278.479} C_VEL
LIN {X 0,Y 535.378,Z 422.154,A -85,B 0,C 180,E1 24277.749,E2 24277.749} C_VEL
LIN {X 0,Y 537.264,Z 425.598,A -85,B 0,C 180,E1 24277.139,E2 24277.139} C_VEL
LIN {X 0,Y 540.589,Z 428.254,A -85,B 0,C 180,E1 24276.22,E2 24276.22} C_VEL
LIN {X 0,Y 543.933,Z 432.885,A -85,B 0,C 180,E1 24275.279,E2 24275.279} C_VEL
LIN {X 0,Y 546.516,Z 435.116,A -85,B 0,C 180,E1 24274.623,E2 24274.623} C_VEL
LIN {X 0,Y 549.609,Z 439.285,A -85,B 0,C 180,E1 24273.821,E2 24273.821} C_VEL
LIN {X 0,Y 551.903,Z 441.509,A -85,B 0,C 180,E1 24273.272,E2 24273.272} C_VEL
LIN {X 0,Y 555.384,Z 445.864,A -85,B 0,C 180,E1 24272.439,E2 24272.439} C_VEL
LIN {X 0,Y 557.244,Z 447.885,A -85,B 0,C 180,E1 24272.016,E2 24272.016} C_VEL
LIN {X 0,Y 562.265,Z 454.05,A -85,B 0,C 180,E1 24270.897,E2 24270.897} C_VEL
LIN {X 0,Y 567.139,Z 460.065,A -85,B 0,C 180,E1 24269.866,E2 24269.866} C_VEL
LIN {X 0,Y 575.144,Z 470.043,A -85,B 0,C 180,E1 24268.271,E2 24268.271} C_VEL
LIN {X 0,Y 586.872,Z 485.448,A -85,B 0,C 180,E1 24266.113,E2 24266.113} C_VEL
LIN {X 0,Y 599.402,Z 502.878,A -85,B 0,C 180,E1 24264.001,E2 24264.001} C_VEL
LIN {X 0,Y 591.521,Z 711.733,A -85,B 0,C 180,E1 24260.923,E2 24260.923} C_VEL
LIN {X 0,Y 585.495,Z 876.246,A -85,B 0,C 180,E1 24258.522,E2 24258.522} C_VEL
LIN {X 0,Y 583.846,Z 900.508,A -85,B 0,C 180,E1 24258.069,E2 24258.069} C_VEL
LIN {X 0,Y 582.042,Z 920.423,A -85,B 0,C 180,E1 24257.586,E2 24257.586} C_VEL
LIN {X 0,Y 580.64,Z 927.948,A -85,B 0,C 180,E1 24257.454,E2 24257.454} C_VEL
LIN {X 0,Y 574.604,Z 946.027,A -85,B 0,C 180,E1 24257.31,E2 24257.31} C_VEL
LIN {X 0,Y 572.813,Z 953.275,A -85,B 0,C 180,E1 24257.143,E2 24257.143} C_VEL
LIN {X 0,Y 572.664,Z 954.299,A -85,B 0,C 180,E1 24257.108,E2 24257.108} C_VEL
LIN {X 0,Y 569.399,Z 977.42,A -85,B 0,C 180,E1 24256.188,E2 24256.188} C_VEL
LIN {X 0,Y 565.068,Z 1004.029,A -85,B 0,C 180,E1 24254.903,E2 24254.903} C_VEL
LIN {X 0,Y 561.46,Z 1024.063,A -85,B 0,C 180,E1 24253.769,E2 24253.769} C_VEL
LIN {X 0,Y 558.017,Z 1041.902,A -85,B 0,C 180,E1 24252.625,E2 24252.625} C_VEL
LIN {X 0,Y 554.433,Z 1059.463,A -85,B 0,C 180,E1 24251.364,E2 24251.364} C_VEL
LIN {X 0,Y 550.631,Z 1077.337,A -85,B 0,C 180,E1 24249.926,E2 24249.926} C_VEL
LIN {X 0,Y 545.978,Z 1098.85,A -85,B 0,C 180,E1 24247.968,E2 24247.968} C_VEL
LIN {X 0,Y 541.503,Z 1118.477,A -85,B 0,C 180,E1 24245.899,E2 24245.899} C_VEL
LIN {X 0,Y 538.073,Z 1133.757,A -85,B 0,C 180,E1 24244.092,E2 24244.092} C_VEL
LIN {X 0,Y 534.855,Z 1148.26,A -85,B 0,C 180,E1 24242.187,E2 24242.187} C_VEL
LIN {X 0,Y 531.141,Z 1166.245,A -85,B 0,C 180,E1 24239.545,E2 24239.545} C_VEL
LIN {X 0,Y 528.16,Z 1181.248,A -85,B 0,C 180,E1 24237.016,E2 24237.016} C_VEL
LIN {X 0,Y 525.98,Z 1193.377,A -85,B 0,C 180,E1 24234.715,E2 24234.715} C_VEL
LIN {X 0,Y 524.217,Z 1204.15,A -85,B 0,C 180,E1 24232.419,E2 24232.419} C_VEL
LIN {X 0,Y 522.56,Z 1215.909,A -85,B 0,C 180,E1 24229.557,E2 24229.557} C_VEL
LIN {X 0,Y 521.414,Z 1225.676,A -85,B 0,C 180,E1 24226.711,E2 24226.711} C_VEL
LIN {X 0,Y 520.754,Z 1232.334,A -85,B 0,C 180,E1 24224.448,E2 24224.448} C_VEL
LIN {X 0,Y 520.361,Z 1237.964,A -85,B 0,C 180,E1 24222.197,E2 24222.197} C_VEL
LIN {X 0,Y 520.083,Z 1242.829,A -85,B 0,C 180,E1 24219.847,E2 24219.847} C_VEL
LIN {X 0,Y 519.964,Z 1246.782,A -85,B 0,C 180,E1 24217.397,E2 24217.397} C_VEL
LIN {X 0,Y 519.92,Z 1249.843,A -85,B 0,C 180,E1 24214.738,E2 24214.738} C_VEL
LIN {X 0,Y 519.908,Z 1251.636,A -85,B 0,C 180,E1 24211.758,E2 24211.758} C_VEL
LIN {X 0,Y 519.865,Z 1251.857,A -85,B 0,C 180,E1 24209.224,E2 24209.224} C_VEL
LIN {X 0,Y 519.91,Z 1251.039,A -85,B 0,C 180,E1 24206.908,E2 24206.908} C_VEL
LIN {X 0,Y 519.926,Z 1249.244,A -85,B 0,C 180,E1 24204.588,E2 24204.588} C_VEL
LIN {X 0,Y 519.967,Z 1246.418,A -85,B 0,C 180,E1 24202.259,E2 24202.259} C_VEL
LIN {X 0,Y 520.121,Z 1242.357,A -85,B 0,C 180,E1 24199.808,E2 24199.808} C_VEL
LIN {X 0,Y 520.462,Z 1236.618,A -85,B 0,C 180,E1 24197.119,E2 24197.119} C_VEL
LIN {X 0,Y 521.155,Z 1228.15,A -85,B 0,C 180,E1 24193.992,E2 24193.992} C_VEL
LIN {X 0,Y 522.063,Z 1219.823,A -85,B 0,C 180,E1 24191.453,E2 24191.453} C_VEL
LIN {X 0,Y 523.265,Z 1210.757,A -85,B 0,C 180,E1 24189.06,E2 24189.06} C_VEL
LIN {X 0,Y 525.011,Z 1199.34,A -85,B 0,C 180,E1 24186.421,E2 24186.421} C_VEL
LIN {X 0,Y 527.511,Z 1184.832,A -85,B 0,C 180,E1 24183.545,E2 24183.545} C_VEL
LIN {X 0,Y 529.87,Z 1172.205,A -85,B 0,C 180,E1 24181.34,E2 24181.34} C_VEL
LIN {X 0,Y 532.541,Z 1159.074,A -85,B 0,C 180,E1 24179.286,E2 24179.286} C_VEL
